(* IEC 61131-3 sources: STVM/tests/functional (part 2) *)

FUNCTION Scale_85 : REAL
VAR_INPUT
    raw : REAL;
END_VAR
    tmp_real := raw * 1.85;
    IF tmp_real > 10000.0 THEN
        tmp_real := 10000.0;
    END_IF;
    Scale_85 := tmp_real;
END_FUNCTION

FUNCTION LimitCheck_85 : BOOL
VAR_INPUT
    value : REAL;
    lo : REAL;
    hi : REAL;
END_VAR
    LimitCheck_85 := (value >= lo) AND (value <= hi);
END_FUNCTION

(* @LOOP_MAX(100) - 校验函数 86 *)
FUNCTION Verify_Channel_86 : INT
VAR_INPUT
    value : REAL;
    limit : REAL;
END_VAR
    tmp_bool := (value <= limit);
    IF tmp_bool THEN
        Verify_Channel_86 := 0;
    ELSE
        Verify_Channel_86 := -1;
    END_IF;
END_FUNCTION

FUNCTION Scale_86 : REAL
VAR_INPUT
    raw : REAL;
END_VAR
    tmp_real := raw * 1.86;
    IF tmp_real > 10000.0 THEN
        tmp_real := 10000.0;
    END_IF;
    Scale_86 := tmp_real;
END_FUNCTION

FUNCTION LimitCheck_86 : BOOL
VAR_INPUT
    value : REAL;
    lo : REAL;
    hi : REAL;
END_VAR
    LimitCheck_86 := (value >= lo) AND (value <= hi);
END_FUNCTION

(* @LOOP_MAX(100) - 校验函数 87 *)
FUNCTION Verify_Channel_87 : INT
VAR_INPUT
    value : REAL;
    limit : REAL;
END_VAR
    tmp_bool := (value <= limit);
    IF tmp_bool THEN
        Verify_Channel_87 := 0;
    ELSE
        Verify_Channel_87 := -1;
    END_IF;
END_FUNCTION

FUNCTION Scale_87 : REAL
VAR_INPUT
    raw : REAL;
END_VAR
    tmp_real := raw * 1.87;
    IF tmp_real > 10000.0 THEN
        tmp_real := 10000.0;
    END_IF;
    Scale_87 := tmp_real;
END_FUNCTION

FUNCTION LimitCheck_87 : BOOL
VAR_INPUT
    value : REAL;
    lo : REAL;
    hi : REAL;
END_VAR
    LimitCheck_87 := (value >= lo) AND (value <= hi);
END_FUNCTION

(* @LOOP_MAX(100) - 校验函数 88 *)
FUNCTION Verify_Channel_88 : INT
VAR_INPUT
    value : REAL;
    limit : REAL;
END_VAR
    tmp_bool := (value <= limit);
    IF tmp_bool THEN
        Verify_Channel_88 := 0;
    ELSE
        Verify_Channel_88 := -1;
    END_IF;
END_FUNCTION

FUNCTION Scale_88 : REAL
VAR_INPUT
    raw : REAL;
END_VAR
    tmp_real := raw * 1.88;
    IF tmp_real > 10000.0 THEN
        tmp_real := 10000.0;
    END_IF;
    Scale_88 := tmp_real;
END_FUNCTION

FUNCTION LimitCheck_88 : BOOL
VAR_INPUT
    value : REAL;
    lo : REAL;
    hi : REAL;
END_VAR
    LimitCheck_88 := (value >= lo) AND (value <= hi);
END_FUNCTION

(* @LOOP_MAX(100) - 校验函数 89 *)
FUNCTION Verify_Channel_89 : INT
VAR_INPUT
    value : REAL;
    limit : REAL;
END_VAR
    tmp_bool := (value <= limit);
    IF tmp_bool THEN
        Verify_Channel_89 := 0;
    ELSE
        Verify_Channel_89 := -1;
    END_IF;
END_FUNCTION

FUNCTION Scale_89 : REAL
VAR_INPUT
    raw : REAL;
END_VAR
    tmp_real := raw * 1.89;
    IF tmp_real > 10000.0 THEN
        tmp_real := 10000.0;
    END_IF;
    Scale_89 := tmp_real;
END_FUNCTION

FUNCTION LimitCheck_89 : BOOL
VAR_INPUT
    value : REAL;
    lo : REAL;
    hi : REAL;
END_VAR
    LimitCheck_89 := (value >= lo) AND (value <= hi);
END_FUNCTION

(* @LOOP_MAX(100) - 校验函数 90 *)
FUNCTION Verify_Channel_90 : INT
VAR_INPUT
    value : REAL;
    limit : REAL;
END_VAR
    tmp_bool := (value <= limit);
    IF tmp_bool THEN
        Verify_Channel_90 := 0;
    ELSE
        Verify_Channel_90 := -1;
    END_IF;
END_FUNCTION

FUNCTION Scale_90 : REAL
VAR_INPUT
    raw : REAL;
END_VAR
    tmp_real := raw * 1.90;
    IF tmp_real > 10000.0 THEN
        tmp_real := 10000.0;
    END_IF;
    Scale_90 := tmp_real;
END_FUNCTION

FUNCTION LimitCheck_90 : BOOL
VAR_INPUT
    value : REAL;
    lo : REAL;
    hi : REAL;
END_VAR
    LimitCheck_90 := (value >= lo) AND (value <= hi);
END_FUNCTION

(* @LOOP_MAX(100) - 校验函数 91 *)
FUNCTION Verify_Channel_91 : INT
VAR_INPUT
    value : REAL;
    limit : REAL;
END_VAR
    tmp_bool := (value <= limit);
    IF tmp_bool THEN
        Verify_Channel_91 := 0;
    ELSE
        Verify_Channel_91 := -1;
    END_IF;
END_FUNCTION

FUNCTION Scale_91 : REAL
VAR_INPUT
    raw : REAL;
END_VAR
    tmp_real := raw * 1.91;
    IF tmp_real > 10000.0 THEN
        tmp_real := 10000.0;
    END_IF;
    Scale_91 := tmp_real;
END_FUNCTION

FUNCTION LimitCheck_91 : BOOL
VAR_INPUT
    value : REAL;
    lo : REAL;
    hi : REAL;
END_VAR
    LimitCheck_91 := (value >= lo) AND (value <= hi);
END_FUNCTION

(* @LOOP_MAX(100) - 校验函数 92 *)
FUNCTION Verify_Channel_92 : INT
VAR_INPUT
    value : REAL;
    limit : REAL;
END_VAR
    tmp_bool := (value <= limit);
    IF tmp_bool THEN
        Verify_Channel_92 := 0;
    ELSE
        Verify_Channel_92 := -1;
    END_IF;
END_FUNCTION

FUNCTION Scale_92 : REAL
VAR_INPUT
    raw : REAL;
END_VAR
    tmp_real := raw * 1.92;
    IF tmp_real > 10000.0 THEN
        tmp_real := 10000.0;
    END_IF;
    Scale_92 := tmp_real;
END_FUNCTION

FUNCTION LimitCheck_92 : BOOL
VAR_INPUT
    value : REAL;
    lo : REAL;
    hi : REAL;
END_VAR
    LimitCheck_92 := (value >= lo) AND (value <= hi);
END_FUNCTION

(* @LOOP_MAX(100) - 校验函数 93 *)
FUNCTION Verify_Channel_93 : INT
VAR_INPUT
    value : REAL;
    limit : REAL;
END_VAR
    tmp_bool := (value <= limit);
    IF tmp_bool THEN
        Verify_Channel_93 := 0;
    ELSE
        Verify_Channel_93 := -1;
    END_IF;
END_FUNCTION

FUNCTION Scale_93 : REAL
VAR_INPUT
    raw : REAL;
END_VAR
    tmp_real := raw * 1.93;
    IF tmp_real > 10000.0 THEN
        tmp_real := 10000.0;
    END_IF;
    Scale_93 := tmp_real;
END_FUNCTION

FUNCTION LimitCheck_93 : BOOL
VAR_INPUT
    value : REAL;
    lo : REAL;
    hi : REAL;
END_VAR
    LimitCheck_93 := (value >= lo) AND (value <= hi);
END_FUNCTION

(* @LOOP_MAX(100) - 校验函数 94 *)
FUNCTION Verify_Channel_94 : INT
VAR_INPUT
    value : REAL;
    limit : REAL;
END_VAR
    tmp_bool := (value <= limit);
    IF tmp_bool THEN
        Verify_Channel_94 := 0;
    ELSE
        Verify_Channel_94 := -1;
    END_IF;
END_FUNCTION

FUNCTION Scale_94 : REAL
VAR_INPUT
    raw : REAL;
END_VAR
    tmp_real := raw * 1.94;
    IF tmp_real > 10000.0 THEN
        tmp_real := 10000.0;
    END_IF;
    Scale_94 := tmp_real;
END_FUNCTION

FUNCTION LimitCheck_94 : BOOL
VAR_INPUT
    value : REAL;
    lo : REAL;
    hi : REAL;
END_VAR
    LimitCheck_94 := (value >= lo) AND (value <= hi);
END_FUNCTION

(* @LOOP_MAX(100) - 校验函数 95 *)
FUNCTION Verify_Channel_95 : INT
VAR_INPUT
    value : REAL;
    limit : REAL;
END_VAR
    tmp_bool := (value <= limit);
    IF tmp_bool THEN
        Verify_Channel_95 := 0;
    ELSE
        Verify_Channel_95 := -1;
    END_IF;
END_FUNCTION

FUNCTION Scale_95 : REAL
VAR_INPUT
    raw : REAL;
END_VAR
    tmp_real := raw * 1.95;
    IF tmp_real > 10000.0 THEN
        tmp_real := 10000.0;
    END_IF;
    Scale_95 := tmp_real;
END_FUNCTION

FUNCTION LimitCheck_95 : BOOL
VAR_INPUT
    value : REAL;
    lo : REAL;
    hi : REAL;
END_VAR
    LimitCheck_95 := (value >= lo) AND (value <= hi);
END_FUNCTION

(* @LOOP_MAX(100) - 校验函数 96 *)
FUNCTION Verify_Channel_96 : INT
VAR_INPUT
    value : REAL;
    limit : REAL;
END_VAR
    tmp_bool := (value <= limit);
    IF tmp_bool THEN
        Verify_Channel_96 := 0;
    ELSE
        Verify_Channel_96 := -1;
    END_IF;
END_FUNCTION

FUNCTION Scale_96 : REAL
VAR_INPUT
    raw : REAL;
END_VAR
    tmp_real := raw * 1.96;
    IF tmp_real > 10000.0 THEN
        tmp_real := 10000.0;
    END_IF;
    Scale_96 := tmp_real;
END_FUNCTION

FUNCTION LimitCheck_96 : BOOL
VAR_INPUT
    value : REAL;
    lo : REAL;
    hi : REAL;
END_VAR
    LimitCheck_96 := (value >= lo) AND (value <= hi);
END_FUNCTION

(* @LOOP_MAX(100) - 校验函数 97 *)
FUNCTION Verify_Channel_97 : INT
VAR_INPUT
    value : REAL;
    limit : REAL;
END_VAR
    tmp_bool := (value <= limit);
    IF tmp_bool THEN
        Verify_Channel_97 := 0;
    ELSE
        Verify_Channel_97 := -1;
    END_IF;
END_FUNCTION

FUNCTION Scale_97 : REAL
VAR_INPUT
    raw : REAL;
END_VAR
    tmp_real := raw * 1.97;
    IF tmp_real > 10000.0 THEN
        tmp_real := 10000.0;
    END_IF;
    Scale_97 := tmp_real;
END_FUNCTION

FUNCTION LimitCheck_97 : BOOL
VAR_INPUT
    value : REAL;
    lo : REAL;
    hi : REAL;
END_VAR
    LimitCheck_97 := (value >= lo) AND (value <= hi);
END_FUNCTION

(* @LOOP_MAX(100) - 校验函数 98 *)
FUNCTION Verify_Channel_98 : INT
VAR_INPUT
    value : REAL;
    limit : REAL;
END_VAR
    tmp_bool := (value <= limit);
    IF tmp_bool THEN
        Verify_Channel_98 := 0;
    ELSE
        Verify_Channel_98 := -1;
    END_IF;
END_FUNCTION

FUNCTION Scale_98 : REAL
VAR_INPUT
    raw : REAL;
END_VAR
    tmp_real := raw * 1.98;
    IF tmp_real > 10000.0 THEN
        tmp_real := 10000.0;
    END_IF;
    Scale_98 := tmp_real;
END_FUNCTION

FUNCTION LimitCheck_98 : BOOL
VAR_INPUT
    value : REAL;
    lo : REAL;
    hi : REAL;
END_VAR
    LimitCheck_98 := (value >= lo) AND (value <= hi);
END_FUNCTION

(* @LOOP_MAX(100) - 校验函数 99 *)
FUNCTION Verify_Channel_99 : INT
VAR_INPUT
    value : REAL;
    limit : REAL;
END_VAR
    tmp_bool := (value <= limit);
    IF tmp_bool THEN
        Verify_Channel_99 := 0;
    ELSE
        Verify_Channel_99 := -1;
    END_IF;
END_FUNCTION

FUNCTION Scale_99 : REAL
VAR_INPUT
    raw : REAL;
END_VAR
    tmp_real := raw * 1.99;
    IF tmp_real > 10000.0 THEN
        tmp_real := 10000.0;
    END_IF;
    Scale_99 := tmp_real;
END_FUNCTION

FUNCTION LimitCheck_99 : BOOL
VAR_INPUT
    value : REAL;
    lo : REAL;
    hi : REAL;
END_VAR
    LimitCheck_99 := (value >= lo) AND (value <= hi);
END_FUNCTION

(* @LOOP_MAX(100) - 校验函数 100 *)
FUNCTION Verify_Channel_100 : INT
VAR_INPUT
    value : REAL;
    limit : REAL;
END_VAR
    tmp_bool := (value <= limit);
    IF tmp_bool THEN
        Verify_Channel_100 := 0;
    ELSE
        Verify_Channel_100 := -1;
    END_IF;
END_FUNCTION

FUNCTION Scale_100 : REAL
VAR_INPUT
    raw : REAL;
END_VAR
    tmp_real := raw * 1.100;
    IF tmp_real > 10000.0 THEN
        tmp_real := 10000.0;
    END_IF;
    Scale_100 := tmp_real;
END_FUNCTION

FUNCTION LimitCheck_100 : BOOL
VAR_INPUT
    value : REAL;
    lo : REAL;
    hi : REAL;
END_VAR
    LimitCheck_100 := (value >= lo) AND (value <= hi);
END_FUNCTION

(* @LOOP_MAX(100) - 校验函数 101 *)
FUNCTION Verify_Channel_101 : INT
VAR_INPUT
    value : REAL;
    limit : REAL;
END_VAR
    tmp_bool := (value <= limit);
    IF tmp_bool THEN
        Verify_Channel_101 := 0;
    ELSE
        Verify_Channel_101 := -1;
    END_IF;
END_FUNCTION

FUNCTION Scale_101 : REAL
VAR_INPUT
    raw : REAL;
END_VAR
    tmp_real := raw * 1.101;
    IF tmp_real > 10000.0 THEN
        tmp_real := 10000.0;
    END_IF;
    Scale_101 := tmp_real;
END_FUNCTION

FUNCTION LimitCheck_101 : BOOL
VAR_INPUT
    value : REAL;
    lo : REAL;
    hi : REAL;
END_VAR
    LimitCheck_101 := (value >= lo) AND (value <= hi);
END_FUNCTION

(* @LOOP_MAX(100) - 校验函数 102 *)
FUNCTION Verify_Channel_102 : INT
VAR_INPUT
    value : REAL;
    limit : REAL;
END_VAR
    tmp_bool := (value <= limit);
    IF tmp_bool THEN
        Verify_Channel_102 := 0;
    ELSE
        Verify_Channel_102 := -1;
    END_IF;
END_FUNCTION

FUNCTION Scale_102 : REAL
VAR_INPUT
    raw : REAL;
END_VAR
    tmp_real := raw * 1.102;
    IF tmp_real > 10000.0 THEN
        tmp_real := 10000.0;
    END_IF;
    Scale_102 := tmp_real;
END_FUNCTION

FUNCTION LimitCheck_102 : BOOL
VAR_INPUT
    value : REAL;
    lo : REAL;
    hi : REAL;
END_VAR
    LimitCheck_102 := (value >= lo) AND (value <= hi);
END_FUNCTION

(* @LOOP_MAX(100) - 校验函数 103 *)
FUNCTION Verify_Channel_103 : INT
VAR_INPUT
    value : REAL;
    limit : REAL;
END_VAR
    tmp_bool := (value <= limit);
    IF tmp_bool THEN
        Verify_Channel_103 := 0;
    ELSE
        Verify_Channel_103 := -1;
    END_IF;
END_FUNCTION

FUNCTION Scale_103 : REAL
VAR_INPUT
    raw : REAL;
END_VAR
    tmp_real := raw * 1.103;
    IF tmp_real > 10000.0 THEN
        tmp_real := 10000.0;
    END_IF;
    Scale_103 := tmp_real;
END_FUNCTION

FUNCTION LimitCheck_103 : BOOL
VAR_INPUT
    value : REAL;
    lo : REAL;
    hi : REAL;
END_VAR
    LimitCheck_103 := (value >= lo) AND (value <= hi);
END_FUNCTION

(* @LOOP_MAX(100) - 校验函数 104 *)
FUNCTION Verify_Channel_104 : INT
VAR_INPUT
    value : REAL;
    limit : REAL;
END_VAR
    tmp_bool := (value <= limit);
    IF tmp_bool THEN
        Verify_Channel_104 := 0;
    ELSE
        Verify_Channel_104 := -1;
    END_IF;
END_FUNCTION

FUNCTION Scale_104 : REAL
VAR_INPUT
    raw : REAL;
END_VAR
    tmp_real := raw * 1.104;
    IF tmp_real > 10000.0 THEN
        tmp_real := 10000.0;
    END_IF;
    Scale_104 := tmp_real;
END_FUNCTION

FUNCTION LimitCheck_104 : BOOL
VAR_INPUT
    value : REAL;
    lo : REAL;
    hi : REAL;
END_VAR
    LimitCheck_104 := (value >= lo) AND (value <= hi);
END_FUNCTION

(* @LOOP_MAX(100) - 校验函数 105 *)
FUNCTION Verify_Channel_105 : INT
VAR_INPUT
    value : REAL;
    limit : REAL;
END_VAR
    tmp_bool := (value <= limit);
    IF tmp_bool THEN
        Verify_Channel_105 := 0;
    ELSE
        Verify_Channel_105 := -1;
    END_IF;
END_FUNCTION

FUNCTION Scale_105 : REAL
VAR_INPUT
    raw : REAL;
END_VAR
    tmp_real := raw * 1.105;
    IF tmp_real > 10000.0 THEN
        tmp_real := 10000.0;
    END_IF;
    Scale_105 := tmp_real;
END_FUNCTION

FUNCTION LimitCheck_105 : BOOL
VAR_INPUT
    value : REAL;
    lo : REAL;
    hi : REAL;
END_VAR
    LimitCheck_105 := (value >= lo) AND (value <= hi);
END_FUNCTION

(* @LOOP_MAX(100) - 校验函数 106 *)
FUNCTION Verify_Channel_106 : INT
VAR_INPUT
    value : REAL;
    limit : REAL;
END_VAR
    tmp_bool := (value <= limit);
    IF tmp_bool THEN
        Verify_Channel_106 := 0;
    ELSE
        Verify_Channel_106 := -1;
    END_IF;
END_FUNCTION

FUNCTION Scale_106 : REAL
VAR_INPUT
    raw : REAL;
END_VAR
    tmp_real := raw * 1.106;
    IF tmp_real > 10000.0 THEN
        tmp_real := 10000.0;
    END_IF;
    Scale_106 := tmp_real;
END_FUNCTION

FUNCTION LimitCheck_106 : BOOL
VAR_INPUT
    value : REAL;
    lo : REAL;
    hi : REAL;
END_VAR
    LimitCheck_106 := (value >= lo) AND (value <= hi);
END_FUNCTION

(* @LOOP_MAX(100) - 校验函数 107 *)
FUNCTION Verify_Channel_107 : INT
VAR_INPUT
    value : REAL;
    limit : REAL;
END_VAR
    tmp_bool := (value <= limit);
    IF tmp_bool THEN
        Verify_Channel_107 := 0;
    ELSE
        Verify_Channel_107 := -1;
    END_IF;
END_FUNCTION

FUNCTION Scale_107 : REAL
VAR_INPUT
    raw : REAL;
END_VAR
    tmp_real := raw * 1.107;
    IF tmp_real > 10000.0 THEN
        tmp_real := 10000.0;
    END_IF;
    Scale_107 := tmp_real;
END_FUNCTION

FUNCTION LimitCheck_107 : BOOL
VAR_INPUT
    value : REAL;
    lo : REAL;
    hi : REAL;
END_VAR
    LimitCheck_107 := (value >= lo) AND (value <= hi);
END_FUNCTION

(* @LOOP_MAX(100) - 校验函数 108 *)
FUNCTION Verify_Channel_108 : INT
VAR_INPUT
    value : REAL;
    limit : REAL;
END_VAR
    tmp_bool := (value <= limit);
    IF tmp_bool THEN
        Verify_Channel_108 := 0;
    ELSE
        Verify_Channel_108 := -1;
    END_IF;
END_FUNCTION

FUNCTION Scale_108 : REAL
VAR_INPUT
    raw : REAL;
END_VAR
    tmp_real := raw * 1.108;
    IF tmp_real > 10000.0 THEN
        tmp_real := 10000.0;
    END_IF;
    Scale_108 := tmp_real;
END_FUNCTION

FUNCTION LimitCheck_108 : BOOL
VAR_INPUT
    value : REAL;
    lo : REAL;
    hi : REAL;
END_VAR
    LimitCheck_108 := (value >= lo) AND (value <= hi);
END_FUNCTION

(* @LOOP_MAX(100) - 校验函数 109 *)
FUNCTION Verify_Channel_109 : INT
VAR_INPUT
    value : REAL;
    limit : REAL;
END_VAR
    tmp_bool := (value <= limit);
    IF tmp_bool THEN
        Verify_Channel_109 := 0;
    ELSE
        Verify_Channel_109 := -1;
    END_IF;
END_FUNCTION

FUNCTION Scale_109 : REAL
VAR_INPUT
    raw : REAL;
END_VAR
    tmp_real := raw * 1.109;
    IF tmp_real > 10000.0 THEN
        tmp_real := 10000.0;
    END_IF;
    Scale_109 := tmp_real;
END_FUNCTION

FUNCTION LimitCheck_109 : BOOL
VAR_INPUT
    value : REAL;
    lo : REAL;
    hi : REAL;
END_VAR
    LimitCheck_109 := (value >= lo) AND (value <= hi);
END_FUNCTION

(* @LOOP_MAX(100) - 校验函数 110 *)
FUNCTION Verify_Channel_110 : INT
VAR_INPUT
    value : REAL;
    limit : REAL;
END_VAR
    tmp_bool := (value <= limit);
    IF tmp_bool THEN
        Verify_Channel_110 := 0;
    ELSE
        Verify_Channel_110 := -1;
    END_IF;
END_FUNCTION

FUNCTION Scale_110 : REAL
VAR_INPUT
    raw : REAL;
END_VAR
    tmp_real := raw * 1.110;
    IF tmp_real > 10000.0 THEN
        tmp_real := 10000.0;
    END_IF;
    Scale_110 := tmp_real;
END_FUNCTION

FUNCTION LimitCheck_110 : BOOL
VAR_INPUT
    value : REAL;
    lo : REAL;
    hi : REAL;
END_VAR
    LimitCheck_110 := (value >= lo) AND (value <= hi);
END_FUNCTION

(* @LOOP_MAX(100) - 校验函数 111 *)
FUNCTION Verify_Channel_111 : INT
VAR_INPUT
    value : REAL;
    limit : REAL;
END_VAR
    tmp_bool := (value <= limit);
    IF tmp_bool THEN
        Verify_Channel_111 := 0;
    ELSE
        Verify_Channel_111 := -1;
    END_IF;
END_FUNCTION

FUNCTION Scale_111 : REAL
VAR_INPUT
    raw : REAL;
END_VAR
    tmp_real := raw * 1.111;
    IF tmp_real > 10000.0 THEN
        tmp_real := 10000.0;
    END_IF;
    Scale_111 := tmp_real;
END_FUNCTION

FUNCTION LimitCheck_111 : BOOL
VAR_INPUT
    value : REAL;
    lo : REAL;
    hi : REAL;
END_VAR
    LimitCheck_111 := (value >= lo) AND (value <= hi);
END_FUNCTION

(* @LOOP_MAX(100) - 校验函数 112 *)
FUNCTION Verify_Channel_112 : INT
VAR_INPUT
    value : REAL;
    limit : REAL;
END_VAR
    tmp_bool := (value <= limit);
    IF tmp_bool THEN
        Verify_Channel_112 := 0;
    ELSE
        Verify_Channel_112 := -1;
    END_IF;
END_FUNCTION

FUNCTION Scale_112 : REAL
VAR_INPUT
    raw : REAL;
END_VAR
    tmp_real := raw * 1.112;
    IF tmp_real > 10000.0 THEN
        tmp_real := 10000.0;
    END_IF;
    Scale_112 := tmp_real;
END_FUNCTION

FUNCTION LimitCheck_112 : BOOL
VAR_INPUT
    value : REAL;
    lo : REAL;
    hi : REAL;
END_VAR
    LimitCheck_112 := (value >= lo) AND (value <= hi);
END_FUNCTION

(* @LOOP_MAX(100) - 校验函数 113 *)
FUNCTION Verify_Channel_113 : INT
VAR_INPUT
    value : REAL;
    limit : REAL;
END_VAR
    tmp_bool := (value <= limit);
    IF tmp_bool THEN
        Verify_Channel_113 := 0;
    ELSE
        Verify_Channel_113 := -1;
    END_IF;
END_FUNCTION

FUNCTION Scale_113 : REAL
VAR_INPUT
    raw : REAL;
END_VAR
    tmp_real := raw * 1.113;
    IF tmp_real > 10000.0 THEN
        tmp_real := 10000.0;
    END_IF;
    Scale_113 := tmp_real;
END_FUNCTION

FUNCTION LimitCheck_113 : BOOL
VAR_INPUT
    value : REAL;
    lo : REAL;
    hi : REAL;
END_VAR
    LimitCheck_113 := (value >= lo) AND (value <= hi);
END_FUNCTION

(* @LOOP_MAX(100) - 校验函数 114 *)
FUNCTION Verify_Channel_114 : INT
VAR_INPUT
    value : REAL;
    limit : REAL;
END_VAR
    tmp_bool := (value <= limit);
    IF tmp_bool THEN
        Verify_Channel_114 := 0;
    ELSE
        Verify_Channel_114 := -1;
    END_IF;
END_FUNCTION

FUNCTION Scale_114 : REAL
VAR_INPUT
    raw : REAL;
END_VAR
    tmp_real := raw * 1.114;
    IF tmp_real > 10000.0 THEN
        tmp_real := 10000.0;
    END_IF;
    Scale_114 := tmp_real;
END_FUNCTION

FUNCTION LimitCheck_114 : BOOL
VAR_INPUT
    value : REAL;
    lo : REAL;
    hi : REAL;
END_VAR
    LimitCheck_114 := (value >= lo) AND (value <= hi);
END_FUNCTION

(* @LOOP_MAX(100) - 校验函数 115 *)
FUNCTION Verify_Channel_115 : INT
VAR_INPUT
    value : REAL;
    limit : REAL;
END_VAR
    tmp_bool := (value <= limit);
    IF tmp_bool THEN
        Verify_Channel_115 := 0;
    ELSE
        Verify_Channel_115 := -1;
    END_IF;
END_FUNCTION

FUNCTION Scale_115 : REAL
VAR_INPUT
    raw : REAL;
END_VAR
    tmp_real := raw * 1.115;
    IF tmp_real > 10000.0 THEN
        tmp_real := 10000.0;
    END_IF;
    Scale_115 := tmp_real;
END_FUNCTION

FUNCTION LimitCheck_115 : BOOL
VAR_INPUT
    value : REAL;
    lo : REAL;
    hi : REAL;
END_VAR
    LimitCheck_115 := (value >= lo) AND (value <= hi);
END_FUNCTION

(* @LOOP_MAX(100) - 校验函数 116 *)
FUNCTION Verify_Channel_116 : INT
VAR_INPUT
    value : REAL;
    limit : REAL;
END_VAR
    tmp_bool := (value <= limit);
    IF tmp_bool THEN
        Verify_Channel_116 := 0;
    ELSE
        Verify_Channel_116 := -1;
    END_IF;
END_FUNCTION

FUNCTION Scale_116 : REAL
VAR_INPUT
    raw : REAL;
END_VAR
    tmp_real := raw * 1.116;
    IF tmp_real > 10000.0 THEN
        tmp_real := 10000.0;
    END_IF;
    Scale_116 := tmp_real;
END_FUNCTION

FUNCTION LimitCheck_116 : BOOL
VAR_INPUT
    value : REAL;
    lo : REAL;
    hi : REAL;
END_VAR
    LimitCheck_116 := (value >= lo) AND (value <= hi);
END_FUNCTION

(* @LOOP_MAX(100) - 校验函数 117 *)
FUNCTION Verify_Channel_117 : INT
VAR_INPUT
    value : REAL;
    limit : REAL;
END_VAR
    tmp_bool := (value <= limit);
    IF tmp_bool THEN
        Verify_Channel_117 := 0;
    ELSE
        Verify_Channel_117 := -1;
    END_IF;
END_FUNCTION

FUNCTION Scale_117 : REAL
VAR_INPUT
    raw : REAL;
END_VAR
    tmp_real := raw * 1.117;
    IF tmp_real > 10000.0 THEN
        tmp_real := 10000.0;
    END_IF;
    Scale_117 := tmp_real;
END_FUNCTION

FUNCTION LimitCheck_117 : BOOL
VAR_INPUT
    value : REAL;
    lo : REAL;
    hi : REAL;
END_VAR
    LimitCheck_117 := (value >= lo) AND (value <= hi);
END_FUNCTION

(* @LOOP_MAX(100) - 校验函数 118 *)
FUNCTION Verify_Channel_118 : INT
VAR_INPUT
    value : REAL;
    limit : REAL;
END_VAR
    tmp_bool := (value <= limit);
    IF tmp_bool THEN
        Verify_Channel_118 := 0;
    ELSE
        Verify_Channel_118 := -1;
    END_IF;
END_FUNCTION

FUNCTION Scale_118 : REAL
VAR_INPUT
    raw : REAL;
END_VAR
    tmp_real := raw * 1.118;
    IF tmp_real > 10000.0 THEN
        tmp_real := 10000.0;
    END_IF;
    Scale_118 := tmp_real;
END_FUNCTION

FUNCTION LimitCheck_118 : BOOL
VAR_INPUT
    value : REAL;
    lo : REAL;
    hi : REAL;
END_VAR
    LimitCheck_118 := (value >= lo) AND (value <= hi);
END_FUNCTION

(* @LOOP_MAX(100) - 校验函数 119 *)
FUNCTION Verify_Channel_119 : INT
VAR_INPUT
    value : REAL;
    limit : REAL;
END_VAR
    tmp_bool := (value <= limit);
    IF tmp_bool THEN
        Verify_Channel_119 := 0;
    ELSE
        Verify_Channel_119 := -1;
    END_IF;
END_FUNCTION

FUNCTION Scale_119 : REAL
VAR_INPUT
    raw : REAL;
END_VAR
    tmp_real := raw * 1.119;
    IF tmp_real > 10000.0 THEN
        tmp_real := 10000.0;
    END_IF;
    Scale_119 := tmp_real;
END_FUNCTION

FUNCTION LimitCheck_119 : BOOL
VAR_INPUT
    value : REAL;
    lo : REAL;
    hi : REAL;
END_VAR
    LimitCheck_119 := (value >= lo) AND (value <= hi);
END_FUNCTION

(* @LOOP_MAX(100) - 校验函数 120 *)
FUNCTION Verify_Channel_120 : INT
VAR_INPUT
    value : REAL;
    limit : REAL;
END_VAR
    tmp_bool := (value <= limit);
    IF tmp_bool THEN
        Verify_Channel_120 := 0;
    ELSE
        Verify_Channel_120 := -1;
    END_IF;
END_FUNCTION

FUNCTION Scale_120 : REAL
VAR_INPUT
    raw : REAL;
END_VAR
    tmp_real := raw * 1.120;
    IF tmp_real > 10000.0 THEN
        tmp_real := 10000.0;
    END_IF;
    Scale_120 := tmp_real;
END_FUNCTION

FUNCTION LimitCheck_120 : BOOL
VAR_INPUT
    value : REAL;
    lo : REAL;
    hi : REAL;
END_VAR
    LimitCheck_120 := (value >= lo) AND (value <= hi);
END_FUNCTION

(* @LOOP_MAX(100) - 校验函数 121 *)
FUNCTION Verify_Channel_121 : INT
VAR_INPUT
    value : REAL;
    limit : REAL;
END_VAR
    tmp_bool := (value <= limit);
    IF tmp_bool THEN
        Verify_Channel_121 := 0;
    ELSE
        Verify_Channel_121 := -1;
    END_IF;
END_FUNCTION

FUNCTION Scale_121 : REAL
VAR_INPUT
    raw : REAL;
END_VAR
    tmp_real := raw * 1.121;
    IF tmp_real > 10000.0 THEN
        tmp_real := 10000.0;
    END_IF;
    Scale_121 := tmp_real;
END_FUNCTION

FUNCTION LimitCheck_121 : BOOL
VAR_INPUT
    value : REAL;
    lo : REAL;
    hi : REAL;
END_VAR
    LimitCheck_121 := (value >= lo) AND (value <= hi);
END_FUNCTION

(* @LOOP_MAX(100) - 校验函数 122 *)
FUNCTION Verify_Channel_122 : INT
VAR_INPUT
    value : REAL;
    limit : REAL;
END_VAR
    tmp_bool := (value <= limit);
    IF tmp_bool THEN
        Verify_Channel_122 := 0;
    ELSE
        Verify_Channel_122 := -1;
    END_IF;
END_FUNCTION

FUNCTION Scale_122 : REAL
VAR_INPUT
    raw : REAL;
END_VAR
    tmp_real := raw * 1.122;
    IF tmp_real > 10000.0 THEN
        tmp_real := 10000.0;
    END_IF;
    Scale_122 := tmp_real;
END_FUNCTION

FUNCTION LimitCheck_122 : BOOL
VAR_INPUT
    value : REAL;
    lo : REAL;
    hi : REAL;
END_VAR
    LimitCheck_122 := (value >= lo) AND (value <= hi);
END_FUNCTION

(* @LOOP_MAX(100) - 校验函数 123 *)
FUNCTION Verify_Channel_123 : INT
VAR_INPUT
    value : REAL;
    limit : REAL;
END_VAR
    tmp_bool := (value <= limit);
    IF tmp_bool THEN
        Verify_Channel_123 := 0;
    ELSE
        Verify_Channel_123 := -1;
    END_IF;
END_FUNCTION

FUNCTION Scale_123 : REAL
VAR_INPUT
    raw : REAL;
END_VAR
    tmp_real := raw * 1.123;
    IF tmp_real > 10000.0 THEN
        tmp_real := 10000.0;
    END_IF;
    Scale_123 := tmp_real;
END_FUNCTION

FUNCTION LimitCheck_123 : BOOL
VAR_INPUT
    value : REAL;
    lo : REAL;
    hi : REAL;
END_VAR
    LimitCheck_123 := (value >= lo) AND (value <= hi);
END_FUNCTION

(* @LOOP_MAX(100) - 校验函数 124 *)
FUNCTION Verify_Channel_124 : INT
VAR_INPUT
    value : REAL;
    limit : REAL;
END_VAR
    tmp_bool := (value <= limit);
    IF tmp_bool THEN
        Verify_Channel_124 := 0;
    ELSE
        Verify_Channel_124 := -1;
    END_IF;
END_FUNCTION

FUNCTION Scale_124 : REAL
VAR_INPUT
    raw : REAL;
END_VAR
    tmp_real := raw * 1.124;
    IF tmp_real > 10000.0 THEN
        tmp_real := 10000.0;
    END_IF;
    Scale_124 := tmp_real;
END_FUNCTION

FUNCTION LimitCheck_124 : BOOL
VAR_INPUT
    value : REAL;
    lo : REAL;
    hi : REAL;
END_VAR
    LimitCheck_124 := (value >= lo) AND (value <= hi);
END_FUNCTION

(* @LOOP_MAX(100) - 校验函数 125 *)
FUNCTION Verify_Channel_125 : INT
VAR_INPUT
    value : REAL;
    limit : REAL;
END_VAR
    tmp_bool := (value <= limit);
    IF tmp_bool THEN
        Verify_Channel_125 := 0;
    ELSE
        Verify_Channel_125 := -1;
    END_IF;
END_FUNCTION

FUNCTION Scale_125 : REAL
VAR_INPUT
    raw : REAL;
END_VAR
    tmp_real := raw * 1.125;
    IF tmp_real > 10000.0 THEN
        tmp_real := 10000.0;
    END_IF;
    Scale_125 := tmp_real;
END_FUNCTION

FUNCTION LimitCheck_125 : BOOL
VAR_INPUT
    value : REAL;
    lo : REAL;
    hi : REAL;
END_VAR
    LimitCheck_125 := (value >= lo) AND (value <= hi);
END_FUNCTION

(* @LOOP_MAX(100) - 校验函数 126 *)
FUNCTION Verify_Channel_126 : INT
VAR_INPUT
    value : REAL;
    limit : REAL;
END_VAR
    tmp_bool := (value <= limit);
    IF tmp_bool THEN
        Verify_Channel_126 := 0;
    ELSE
        Verify_Channel_126 := -1;
    END_IF;
END_FUNCTION

FUNCTION Scale_126 : REAL
VAR_INPUT
    raw : REAL;
END_VAR
    tmp_real := raw * 1.126;
    IF tmp_real > 10000.0 THEN
        tmp_real := 10000.0;
    END_IF;
    Scale_126 := tmp_real;
END_FUNCTION

FUNCTION LimitCheck_126 : BOOL
VAR_INPUT
    value : REAL;
    lo : REAL;
    hi : REAL;
END_VAR
    LimitCheck_126 := (value >= lo) AND (value <= hi);
END_FUNCTION

(* @LOOP_MAX(100) - 校验函数 127 *)
FUNCTION Verify_Channel_127 : INT
VAR_INPUT
    value : REAL;
    limit : REAL;
END_VAR
    tmp_bool := (value <= limit);
    IF tmp_bool THEN
        Verify_Channel_127 := 0;
    ELSE
        Verify_Channel_127 := -1;
    END_IF;
END_FUNCTION

FUNCTION Scale_127 : REAL
VAR_INPUT
    raw : REAL;
END_VAR
    tmp_real := raw * 1.127;
    IF tmp_real > 10000.0 THEN
        tmp_real := 10000.0;
    END_IF;
    Scale_127 := tmp_real;
END_FUNCTION

FUNCTION LimitCheck_127 : BOOL
VAR_INPUT
    value : REAL;
    lo : REAL;
    hi : REAL;
END_VAR
    LimitCheck_127 := (value >= lo) AND (value <= hi);
END_FUNCTION

(* @LOOP_MAX(100) - 校验函数 128 *)
FUNCTION Verify_Channel_128 : INT
VAR_INPUT
    value : REAL;
    limit : REAL;
END_VAR
    tmp_bool := (value <= limit);
    IF tmp_bool THEN
        Verify_Channel_128 := 0;
    ELSE
        Verify_Channel_128 := -1;
    END_IF;
END_FUNCTION

FUNCTION Scale_128 : REAL
VAR_INPUT
    raw : REAL;
END_VAR
    tmp_real := raw * 1.128;
    IF tmp_real > 10000.0 THEN
        tmp_real := 10000.0;
    END_IF;
    Scale_128 := tmp_real;
END_FUNCTION

FUNCTION LimitCheck_128 : BOOL
VAR_INPUT
    value : REAL;
    lo : REAL;
    hi : REAL;
END_VAR
    LimitCheck_128 := (value >= lo) AND (value <= hi);
END_FUNCTION

(* @LOOP_MAX(100) - 校验函数 129 *)
FUNCTION Verify_Channel_129 : INT
VAR_INPUT
    value : REAL;
    limit : REAL;
END_VAR
    tmp_bool := (value <= limit);
    IF tmp_bool THEN
        Verify_Channel_129 := 0;
    ELSE
        Verify_Channel_129 := -1;
    END_IF;
END_FUNCTION

FUNCTION Scale_129 : REAL
VAR_INPUT
    raw : REAL;
END_VAR
    tmp_real := raw * 1.129;
    IF tmp_real > 10000.0 THEN
        tmp_real := 10000.0;
    END_IF;
    Scale_129 := tmp_real;
END_FUNCTION

FUNCTION LimitCheck_129 : BOOL
VAR_INPUT
    value : REAL;
    lo : REAL;
    hi : REAL;
END_VAR
    LimitCheck_129 := (value >= lo) AND (value <= hi);
END_FUNCTION

(* @LOOP_MAX(100) - 校验函数 130 *)
FUNCTION Verify_Channel_130 : INT
VAR_INPUT
    value : REAL;
    limit : REAL;
END_VAR
    tmp_bool := (value <= limit);
    IF tmp_bool THEN
        Verify_Channel_130 := 0;
    ELSE
        Verify_Channel_130 := -1;
    END_IF;
END_FUNCTION

FUNCTION Scale_130 : REAL
VAR_INPUT
    raw : REAL;
END_VAR
    tmp_real := raw * 1.130;
    IF tmp_real > 10000.0 THEN
        tmp_real := 10000.0;
    END_IF;
    Scale_130 := tmp_real;
END_FUNCTION

FUNCTION LimitCheck_130 : BOOL
VAR_INPUT
    value : REAL;
    lo : REAL;
    hi : REAL;
END_VAR
    LimitCheck_130 := (value >= lo) AND (value <= hi);
END_FUNCTION

(* @LOOP_MAX(100) - 校验函数 131 *)
FUNCTION Verify_Channel_131 : INT
VAR_INPUT
    value : REAL;
    limit : REAL;
END_VAR
    tmp_bool := (value <= limit);
    IF tmp_bool THEN
        Verify_Channel_131 := 0;
    ELSE
        Verify_Channel_131 := -1;
    END_IF;
END_FUNCTION

FUNCTION Scale_131 : REAL
VAR_INPUT
    raw : REAL;
END_VAR
    tmp_real := raw * 1.131;
    IF tmp_real > 10000.0 THEN
        tmp_real := 10000.0;
    END_IF;
    Scale_131 := tmp_real;
END_FUNCTION

FUNCTION LimitCheck_131 : BOOL
VAR_INPUT
    value : REAL;
    lo : REAL;
    hi : REAL;
END_VAR
    LimitCheck_131 := (value >= lo) AND (value <= hi);
END_FUNCTION

(* @LOOP_MAX(100) - 校验函数 132 *)
FUNCTION Verify_Channel_132 : INT
VAR_INPUT
    value : REAL;
    limit : REAL;
END_VAR
    tmp_bool := (value <= limit);
    IF tmp_bool THEN
        Verify_Channel_132 := 0;
    ELSE
        Verify_Channel_132 := -1;
    END_IF;
END_FUNCTION

FUNCTION Scale_132 : REAL
VAR_INPUT
    raw : REAL;
END_VAR
    tmp_real := raw * 1.132;
    IF tmp_real > 10000.0 THEN
        tmp_real := 10000.0;
    END_IF;
    Scale_132 := tmp_real;
END_FUNCTION

FUNCTION LimitCheck_132 : BOOL
VAR_INPUT
    value : REAL;
    lo : REAL;
    hi : REAL;
END_VAR
    LimitCheck_132 := (value >= lo) AND (value <= hi);
END_FUNCTION

(* @LOOP_MAX(100) - 校验函数 133 *)
FUNCTION Verify_Channel_133 : INT
VAR_INPUT
    value : REAL;
    limit : REAL;
END_VAR
    tmp_bool := (value <= limit);
    IF tmp_bool THEN
        Verify_Channel_133 := 0;
    ELSE
        Verify_Channel_133 := -1;
    END_IF;
END_FUNCTION

FUNCTION Scale_133 : REAL
VAR_INPUT
    raw : REAL;
END_VAR
    tmp_real := raw * 1.133;
    IF tmp_real > 10000.0 THEN
        tmp_real := 10000.0;
    END_IF;
    Scale_133 := tmp_real;
END_FUNCTION

FUNCTION LimitCheck_133 : BOOL
VAR_INPUT
    value : REAL;
    lo : REAL;
    hi : REAL;
END_VAR
    LimitCheck_133 := (value >= lo) AND (value <= hi);
END_FUNCTION

(* @LOOP_MAX(100) - 校验函数 134 *)
FUNCTION Verify_Channel_134 : INT
VAR_INPUT
    value : REAL;
    limit : REAL;
END_VAR
    tmp_bool := (value <= limit);
    IF tmp_bool THEN
        Verify_Channel_134 := 0;
    ELSE
        Verify_Channel_134 := -1;
    END_IF;
END_FUNCTION

FUNCTION Scale_134 : REAL
VAR_INPUT
    raw : REAL;
END_VAR
    tmp_real := raw * 1.134;
    IF tmp_real > 10000.0 THEN
        tmp_real := 10000.0;
    END_IF;
    Scale_134 := tmp_real;
END_FUNCTION

FUNCTION LimitCheck_134 : BOOL
VAR_INPUT
    value : REAL;
    lo : REAL;
    hi : REAL;
END_VAR
    LimitCheck_134 := (value >= lo) AND (value <= hi);
END_FUNCTION

(* @LOOP_MAX(100) - 校验函数 135 *)
FUNCTION Verify_Channel_135 : INT
VAR_INPUT
    value : REAL;
    limit : REAL;
END_VAR
    tmp_bool := (value <= limit);
    IF tmp_bool THEN
        Verify_Channel_135 := 0;
    ELSE
        Verify_Channel_135 := -1;
    END_IF;
END_FUNCTION

FUNCTION Scale_135 : REAL
VAR_INPUT
    raw : REAL;
END_VAR
    tmp_real := raw * 1.135;
    IF tmp_real > 10000.0 THEN
        tmp_real := 10000.0;
    END_IF;
    Scale_135 := tmp_real;
END_FUNCTION

FUNCTION LimitCheck_135 : BOOL
VAR_INPUT
    value : REAL;
    lo : REAL;
    hi : REAL;
END_VAR
    LimitCheck_135 := (value >= lo) AND (value <= hi);
END_FUNCTION

(* @LOOP_MAX(100) - 校验函数 136 *)
FUNCTION Verify_Channel_136 : INT
VAR_INPUT
    value : REAL;
    limit : REAL;
END_VAR
    tmp_bool := (value <= limit);
    IF tmp_bool THEN
        Verify_Channel_136 := 0;
    ELSE
        Verify_Channel_136 := -1;
    END_IF;
END_FUNCTION

FUNCTION Scale_136 : REAL
VAR_INPUT
    raw : REAL;
END_VAR
    tmp_real := raw * 1.136;
    IF tmp_real > 10000.0 THEN
        tmp_real := 10000.0;
    END_IF;
    Scale_136 := tmp_real;
END_FUNCTION

FUNCTION LimitCheck_136 : BOOL
VAR_INPUT
    value : REAL;
    lo : REAL;
    hi : REAL;
END_VAR
    LimitCheck_136 := (value >= lo) AND (value <= hi);
END_FUNCTION

(* @LOOP_MAX(100) - 校验函数 137 *)
FUNCTION Verify_Channel_137 : INT
VAR_INPUT
    value : REAL;
    limit : REAL;
END_VAR
    tmp_bool := (value <= limit);
    IF tmp_bool THEN
        Verify_Channel_137 := 0;
    ELSE
        Verify_Channel_137 := -1;
    END_IF;
END_FUNCTION

FUNCTION Scale_137 : REAL
VAR_INPUT
    raw : REAL;
END_VAR
    tmp_real := raw * 1.137;
    IF tmp_real > 10000.0 THEN
        tmp_real := 10000.0;
    END_IF;
    Scale_137 := tmp_real;
END_FUNCTION

FUNCTION LimitCheck_137 : BOOL
VAR_INPUT
    value : REAL;
    lo : REAL;
    hi : REAL;
END_VAR
    LimitCheck_137 := (value >= lo) AND (value <= hi);
END_FUNCTION

(* @LOOP_MAX(100) - 校验函数 138 *)
FUNCTION Verify_Channel_138 : INT
VAR_INPUT
    value : REAL;
    limit : REAL;
END_VAR
    tmp_bool := (value <= limit);
    IF tmp_bool THEN
        Verify_Channel_138 := 0;
    ELSE
        Verify_Channel_138 := -1;
    END_IF;
END_FUNCTION

FUNCTION Scale_138 : REAL
VAR_INPUT
    raw : REAL;
END_VAR
    tmp_real := raw * 1.138;
    IF tmp_real > 10000.0 THEN
        tmp_real := 10000.0;
    END_IF;
    Scale_138 := tmp_real;
END_FUNCTION

FUNCTION LimitCheck_138 : BOOL
VAR_INPUT
    value : REAL;
    lo : REAL;
    hi : REAL;
END_VAR
    LimitCheck_138 := (value >= lo) AND (value <= hi);
END_FUNCTION

(* @LOOP_MAX(100) - 校验函数 139 *)
FUNCTION Verify_Channel_139 : INT
VAR_INPUT
    value : REAL;
    limit : REAL;
END_VAR
    tmp_bool := (value <= limit);
    IF tmp_bool THEN
        Verify_Channel_139 := 0;
    ELSE
        Verify_Channel_139 := -1;
    END_IF;
END_FUNCTION

FUNCTION Scale_139 : REAL
VAR_INPUT
    raw : REAL;
END_VAR
    tmp_real := raw * 1.139;
    IF tmp_real > 10000.0 THEN
        tmp_real := 10000.0;
    END_IF;
    Scale_139 := tmp_real;
END_FUNCTION

FUNCTION LimitCheck_139 : BOOL
VAR_INPUT
    value : REAL;
    lo : REAL;
    hi : REAL;
END_VAR
    LimitCheck_139 := (value >= lo) AND (value <= hi);
END_FUNCTION

(* @LOOP_MAX(100) - 校验函数 140 *)
FUNCTION Verify_Channel_140 : INT
VAR_INPUT
    value : REAL;
    limit : REAL;
END_VAR
    tmp_bool := (value <= limit);
    IF tmp_bool THEN
        Verify_Channel_140 := 0;
    ELSE
        Verify_Channel_140 := -1;
    END_IF;
END_FUNCTION

FUNCTION Scale_140 : REAL
VAR_INPUT
    raw : REAL;
END_VAR
    tmp_real := raw * 1.140;
    IF tmp_real > 10000.0 THEN
        tmp_real := 10000.0;
    END_IF;
    Scale_140 := tmp_real;
END_FUNCTION

FUNCTION LimitCheck_140 : BOOL
VAR_INPUT
    value : REAL;
    lo : REAL;
    hi : REAL;
END_VAR
    LimitCheck_140 := (value >= lo) AND (value <= hi);
END_FUNCTION

(* @LOOP_MAX(100) - 校验函数 141 *)
FUNCTION Verify_Channel_141 : INT
VAR_INPUT
    value : REAL;
    limit : REAL;
END_VAR
    tmp_bool := (value <= limit);
    IF tmp_bool THEN
        Verify_Channel_141 := 0;
    ELSE
        Verify_Channel_141 := -1;
    END_IF;
END_FUNCTION

FUNCTION Scale_141 : REAL
VAR_INPUT
    raw : REAL;
END_VAR
    tmp_real := raw * 1.141;
    IF tmp_real > 10000.0 THEN
        tmp_real := 10000.0;
    END_IF;
    Scale_141 := tmp_real;
END_FUNCTION

FUNCTION LimitCheck_141 : BOOL
VAR_INPUT
    value : REAL;
    lo : REAL;
    hi : REAL;
END_VAR
    LimitCheck_141 := (value >= lo) AND (value <= hi);
END_FUNCTION

(* @LOOP_MAX(100) - 校验函数 142 *)
FUNCTION Verify_Channel_142 : INT
VAR_INPUT
    value : REAL;
    limit : REAL;
END_VAR
    tmp_bool := (value <= limit);
    IF tmp_bool THEN
        Verify_Channel_142 := 0;
    ELSE
        Verify_Channel_142 := -1;
    END_IF;
END_FUNCTION

FUNCTION Scale_142 : REAL
VAR_INPUT
    raw : REAL;
END_VAR
    tmp_real := raw * 1.142;
    IF tmp_real > 10000.0 THEN
        tmp_real := 10000.0;
    END_IF;
    Scale_142 := tmp_real;
END_FUNCTION

FUNCTION LimitCheck_142 : BOOL
VAR_INPUT
    value : REAL;
    lo : REAL;
    hi : REAL;
END_VAR
    LimitCheck_142 := (value >= lo) AND (value <= hi);
END_FUNCTION

(* @LOOP_MAX(100) - 校验函数 143 *)
FUNCTION Verify_Channel_143 : INT
VAR_INPUT
    value : REAL;
    limit : REAL;
END_VAR
    tmp_bool := (value <= limit);
    IF tmp_bool THEN
        Verify_Channel_143 := 0;
    ELSE
        Verify_Channel_143 := -1;
    END_IF;
END_FUNCTION

FUNCTION Scale_143 : REAL
VAR_INPUT
    raw : REAL;
END_VAR
    tmp_real := raw * 1.143;
    IF tmp_real > 10000.0 THEN
        tmp_real := 10000.0;
    END_IF;
    Scale_143 := tmp_real;
END_FUNCTION

FUNCTION LimitCheck_143 : BOOL
VAR_INPUT
    value : REAL;
    lo : REAL;
    hi : REAL;
END_VAR
    LimitCheck_143 := (value >= lo) AND (value <= hi);
END_FUNCTION

(* @LOOP_MAX(100) - 校验函数 144 *)
FUNCTION Verify_Channel_144 : INT
VAR_INPUT
    value : REAL;
    limit : REAL;
END_VAR
    tmp_bool := (value <= limit);
    IF tmp_bool THEN
        Verify_Channel_144 := 0;
    ELSE
        Verify_Channel_144 := -1;
    END_IF;
END_FUNCTION

FUNCTION Scale_144 : REAL
VAR_INPUT
    raw : REAL;
END_VAR
    tmp_real := raw * 1.144;
    IF tmp_real > 10000.0 THEN
        tmp_real := 10000.0;
    END_IF;
    Scale_144 := tmp_real;
END_FUNCTION

FUNCTION LimitCheck_144 : BOOL
VAR_INPUT
    value : REAL;
    lo : REAL;
    hi : REAL;
END_VAR
    LimitCheck_144 := (value >= lo) AND (value <= hi);
END_FUNCTION

(* @LOOP_MAX(100) - 校验函数 145 *)
FUNCTION Verify_Channel_145 : INT
VAR_INPUT
    value : REAL;
    limit : REAL;
END_VAR
    tmp_bool := (value <= limit);
    IF tmp_bool THEN
        Verify_Channel_145 := 0;
    ELSE
        Verify_Channel_145 := -1;
    END_IF;
END_FUNCTION

FUNCTION Scale_145 : REAL
VAR_INPUT
    raw : REAL;
END_VAR
    tmp_real := raw * 1.145;
    IF tmp_real > 10000.0 THEN
        tmp_real := 10000.0;
    END_IF;
    Scale_145 := tmp_real;
END_FUNCTION

FUNCTION LimitCheck_145 : BOOL
VAR_INPUT
    value : REAL;
    lo : REAL;
    hi : REAL;
END_VAR
    LimitCheck_145 := (value >= lo) AND (value <= hi);
END_FUNCTION

(* @LOOP_MAX(100) - 校验函数 146 *)
FUNCTION Verify_Channel_146 : INT
VAR_INPUT
    value : REAL;
    limit : REAL;
END_VAR
    tmp_bool := (value <= limit);
    IF tmp_bool THEN
        Verify_Channel_146 := 0;
    ELSE
        Verify_Channel_146 := -1;
    END_IF;
END_FUNCTION

FUNCTION Scale_146 : REAL
VAR_INPUT
    raw : REAL;
END_VAR
    tmp_real := raw * 1.146;
    IF tmp_real > 10000.0 THEN
        tmp_real := 10000.0;
    END_IF;
    Scale_146 := tmp_real;
END_FUNCTION

FUNCTION LimitCheck_146 : BOOL
VAR_INPUT
    value : REAL;
    lo : REAL;
    hi : REAL;
END_VAR
    LimitCheck_146 := (value >= lo) AND (value <= hi);
END_FUNCTION

(* @LOOP_MAX(100) - 校验函数 147 *)
FUNCTION Verify_Channel_147 : INT
VAR_INPUT
    value : REAL;
    limit : REAL;
END_VAR
    tmp_bool := (value <= limit);
    IF tmp_bool THEN
        Verify_Channel_147 := 0;
    ELSE
        Verify_Channel_147 := -1;
    END_IF;
END_FUNCTION

FUNCTION Scale_147 : REAL
VAR_INPUT
    raw : REAL;
END_VAR
    tmp_real := raw * 1.147;
    IF tmp_real > 10000.0 THEN
        tmp_real := 10000.0;
    END_IF;
    Scale_147 := tmp_real;
END_FUNCTION

FUNCTION LimitCheck_147 : BOOL
VAR_INPUT
    value : REAL;
    lo : REAL;
    hi : REAL;
END_VAR
    LimitCheck_147 := (value >= lo) AND (value <= hi);
END_FUNCTION

(* @LOOP_MAX(100) - 校验函数 148 *)
FUNCTION Verify_Channel_148 : INT
VAR_INPUT
    value : REAL;
    limit : REAL;
END_VAR
    tmp_bool := (value <= limit);
    IF tmp_bool THEN
        Verify_Channel_148 := 0;
    ELSE
        Verify_Channel_148 := -1;
    END_IF;
END_FUNCTION

FUNCTION Scale_148 : REAL
VAR_INPUT
    raw : REAL;
END_VAR
    tmp_real := raw * 1.148;
    IF tmp_real > 10000.0 THEN
        tmp_real := 10000.0;
    END_IF;
    Scale_148 := tmp_real;
END_FUNCTION

FUNCTION LimitCheck_148 : BOOL
VAR_INPUT
    value : REAL;
    lo : REAL;
    hi : REAL;
END_VAR
    LimitCheck_148 := (value >= lo) AND (value <= hi);
END_FUNCTION

(* @LOOP_MAX(100) - 校验函数 149 *)
FUNCTION Verify_Channel_149 : INT
VAR_INPUT
    value : REAL;
    limit : REAL;
END_VAR
    tmp_bool := (value <= limit);
    IF tmp_bool THEN
        Verify_Channel_149 := 0;
    ELSE
        Verify_Channel_149 := -1;
    END_IF;
END_FUNCTION

FUNCTION Scale_149 : REAL
VAR_INPUT
    raw : REAL;
END_VAR
    tmp_real := raw * 1.149;
    IF tmp_real > 10000.0 THEN
        tmp_real := 10000.0;
    END_IF;
    Scale_149 := tmp_real;
END_FUNCTION

FUNCTION LimitCheck_149 : BOOL
VAR_INPUT
    value : REAL;
    lo : REAL;
    hi : REAL;
END_VAR
    LimitCheck_149 := (value >= lo) AND (value <= hi);
END_FUNCTION

(* @LOOP_MAX(100) - 校验函数 150 *)
FUNCTION Verify_Channel_150 : INT
VAR_INPUT
    value : REAL;
    limit : REAL;
END_VAR
    tmp_bool := (value <= limit);
    IF tmp_bool THEN
        Verify_Channel_150 := 0;
    ELSE
        Verify_Channel_150 := -1;
    END_IF;
END_FUNCTION

FUNCTION Scale_150 : REAL
VAR_INPUT
    raw : REAL;
END_VAR
    tmp_real := raw * 1.150;
    IF tmp_real > 10000.0 THEN
        tmp_real := 10000.0;
    END_IF;
    Scale_150 := tmp_real;
END_FUNCTION

FUNCTION LimitCheck_150 : BOOL
VAR_INPUT
    value : REAL;
    lo : REAL;
    hi : REAL;
END_VAR
    LimitCheck_150 := (value >= lo) AND (value <= hi);
END_FUNCTION

(* @LOOP_MAX(100) - 校验函数 151 *)
FUNCTION Verify_Channel_151 : INT
VAR_INPUT
    value : REAL;
    limit : REAL;
END_VAR
    tmp_bool := (value <= limit);
    IF tmp_bool THEN
        Verify_Channel_151 := 0;
    ELSE
        Verify_Channel_151 := -1;
    END_IF;
END_FUNCTION

FUNCTION Scale_151 : REAL
VAR_INPUT
    raw : REAL;
END_VAR
    tmp_real := raw * 1.151;
    IF tmp_real > 10000.0 THEN
        tmp_real := 10000.0;
    END_IF;
    Scale_151 := tmp_real;
END_FUNCTION

FUNCTION LimitCheck_151 : BOOL
VAR_INPUT
    value : REAL;
    lo : REAL;
    hi : REAL;
END_VAR
    LimitCheck_151 := (value >= lo) AND (value <= hi);
END_FUNCTION

(* @LOOP_MAX(100) - 校验函数 152 *)
FUNCTION Verify_Channel_152 : INT
VAR_INPUT
    value : REAL;
    limit : REAL;
END_VAR
    tmp_bool := (value <= limit);
    IF tmp_bool THEN
        Verify_Channel_152 := 0;
    ELSE
        Verify_Channel_152 := -1;
    END_IF;
END_FUNCTION

FUNCTION Scale_152 : REAL
VAR_INPUT
    raw : REAL;
END_VAR
    tmp_real := raw * 1.152;
    IF tmp_real > 10000.0 THEN
        tmp_real := 10000.0;
    END_IF;
    Scale_152 := tmp_real;
END_FUNCTION

FUNCTION LimitCheck_152 : BOOL
VAR_INPUT
    value : REAL;
    lo : REAL;
    hi : REAL;
END_VAR
    LimitCheck_152 := (value >= lo) AND (value <= hi);
END_FUNCTION

(* @LOOP_MAX(100) - 校验函数 153 *)
FUNCTION Verify_Channel_153 : INT
VAR_INPUT
    value : REAL;
    limit : REAL;
END_VAR
    tmp_bool := (value <= limit);
    IF tmp_bool THEN
        Verify_Channel_153 := 0;
    ELSE
        Verify_Channel_153 := -1;
    END_IF;
END_FUNCTION

FUNCTION Scale_153 : REAL
VAR_INPUT
    raw : REAL;
END_VAR
    tmp_real := raw * 1.153;
    IF tmp_real > 10000.0 THEN
        tmp_real := 10000.0;
    END_IF;
    Scale_153 := tmp_real;
END_FUNCTION

FUNCTION LimitCheck_153 : BOOL
VAR_INPUT
    value : REAL;
    lo : REAL;
    hi : REAL;
END_VAR
    LimitCheck_153 := (value >= lo) AND (value <= hi);
END_FUNCTION

(* @LOOP_MAX(100) - 校验函数 154 *)
FUNCTION Verify_Channel_154 : INT
VAR_INPUT
    value : REAL;
    limit : REAL;
END_VAR
    tmp_bool := (value <= limit);
    IF tmp_bool THEN
        Verify_Channel_154 := 0;
    ELSE
        Verify_Channel_154 := -1;
    END_IF;
END_FUNCTION

FUNCTION Scale_154 : REAL
VAR_INPUT
    raw : REAL;
END_VAR
    tmp_real := raw * 1.154;
    IF tmp_real > 10000.0 THEN
        tmp_real := 10000.0;
    END_IF;
    Scale_154 := tmp_real;
END_FUNCTION

FUNCTION LimitCheck_154 : BOOL
VAR_INPUT
    value : REAL;
    lo : REAL;
    hi : REAL;
END_VAR
    LimitCheck_154 := (value >= lo) AND (value <= hi);
END_FUNCTION

(* @LOOP_MAX(100) - 校验函数 155 *)
FUNCTION Verify_Channel_155 : INT
VAR_INPUT
    value : REAL;
    limit : REAL;
END_VAR
    tmp_bool := (value <= limit);
    IF tmp_bool THEN
        Verify_Channel_155 := 0;
    ELSE
        Verify_Channel_155 := -1;
    END_IF;
END_FUNCTION

FUNCTION Scale_155 : REAL
VAR_INPUT
    raw : REAL;
END_VAR
    tmp_real := raw * 1.155;
    IF tmp_real > 10000.0 THEN
        tmp_real := 10000.0;
    END_IF;
    Scale_155 := tmp_real;
END_FUNCTION

FUNCTION LimitCheck_155 : BOOL
VAR_INPUT
    value : REAL;
    lo : REAL;
    hi : REAL;
END_VAR
    LimitCheck_155 := (value >= lo) AND (value <= hi);
END_FUNCTION

(* @LOOP_MAX(100) - 校验函数 156 *)
FUNCTION Verify_Channel_156 : INT
VAR_INPUT
    value : REAL;
    limit : REAL;
END_VAR
    tmp_bool := (value <= limit);
    IF tmp_bool THEN
        Verify_Channel_156 := 0;
    ELSE
        Verify_Channel_156 := -1;
    END_IF;
END_FUNCTION

FUNCTION Scale_156 : REAL
VAR_INPUT
    raw : REAL;
END_VAR
    tmp_real := raw * 1.156;
    IF tmp_real > 10000.0 THEN
        tmp_real := 10000.0;
    END_IF;
    Scale_156 := tmp_real;
END_FUNCTION

FUNCTION LimitCheck_156 : BOOL
VAR_INPUT
    value : REAL;
    lo : REAL;
    hi : REAL;
END_VAR
    LimitCheck_156 := (value >= lo) AND (value <= hi);
END_FUNCTION

(* @LOOP_MAX(100) - 校验函数 157 *)
FUNCTION Verify_Channel_157 : INT
VAR_INPUT
    value : REAL;
    limit : REAL;
END_VAR
    tmp_bool := (value <= limit);
    IF tmp_bool THEN
        Verify_Channel_157 := 0;
    ELSE
        Verify_Channel_157 := -1;
    END_IF;
END_FUNCTION

FUNCTION Scale_157 : REAL
VAR_INPUT
    raw : REAL;
END_VAR
    tmp_real := raw * 1.157;
    IF tmp_real > 10000.0 THEN
        tmp_real := 10000.0;
    END_IF;
    Scale_157 := tmp_real;
END_FUNCTION

FUNCTION LimitCheck_157 : BOOL
VAR_INPUT
    value : REAL;
    lo : REAL;
    hi : REAL;
END_VAR
    LimitCheck_157 := (value >= lo) AND (value <= hi);
END_FUNCTION

(* @LOOP_MAX(100) - 校验函数 158 *)
FUNCTION Verify_Channel_158 : INT
VAR_INPUT
    value : REAL;
    limit : REAL;
END_VAR
    tmp_bool := (value <= limit);
    IF tmp_bool THEN
        Verify_Channel_158 := 0;
    ELSE
        Verify_Channel_158 := -1;
    END_IF;
END_FUNCTION

FUNCTION Scale_158 : REAL
VAR_INPUT
    raw : REAL;
END_VAR
    tmp_real := raw * 1.158;
    IF tmp_real > 10000.0 THEN
        tmp_real := 10000.0;
    END_IF;
    Scale_158 := tmp_real;
END_FUNCTION

FUNCTION LimitCheck_158 : BOOL
VAR_INPUT
    value : REAL;
    lo : REAL;
    hi : REAL;
END_VAR
    LimitCheck_158 := (value >= lo) AND (value <= hi);
END_FUNCTION

(* @LOOP_MAX(100) - 校验函数 159 *)
FUNCTION Verify_Channel_159 : INT
VAR_INPUT
    value : REAL;
    limit : REAL;
END_VAR
    tmp_bool := (value <= limit);
    IF tmp_bool THEN
        Verify_Channel_159 := 0;
    ELSE
        Verify_Channel_159 := -1;
    END_IF;
END_FUNCTION

FUNCTION Scale_159 : REAL
VAR_INPUT
    raw : REAL;
END_VAR
    tmp_real := raw * 1.159;
    IF tmp_real > 10000.0 THEN
        tmp_real := 10000.0;
    END_IF;
    Scale_159 := tmp_real;
END_FUNCTION

FUNCTION LimitCheck_159 : BOOL
VAR_INPUT
    value : REAL;
    lo : REAL;
    hi : REAL;
END_VAR
    LimitCheck_159 := (value >= lo) AND (value <= hi);
END_FUNCTION

(* @LOOP_MAX(100) - 校验函数 160 *)
FUNCTION Verify_Channel_160 : INT
VAR_INPUT
    value : REAL;
    limit : REAL;
END_VAR
    tmp_bool := (value <= limit);
    IF tmp_bool THEN
        Verify_Channel_160 := 0;
    ELSE
        Verify_Channel_160 := -1;
    END_IF;
END_FUNCTION

FUNCTION Scale_160 : REAL
VAR_INPUT
    raw : REAL;
END_VAR
    tmp_real := raw * 1.160;
    IF tmp_real > 10000.0 THEN
        tmp_real := 10000.0;
    END_IF;
    Scale_160 := tmp_real;
END_FUNCTION

FUNCTION LimitCheck_160 : BOOL
VAR_INPUT
    value : REAL;
    lo : REAL;
    hi : REAL;
END_VAR
    LimitCheck_160 := (value >= lo) AND (value <= hi);
END_FUNCTION

(* @LOOP_MAX(100) - 校验函数 161 *)
FUNCTION Verify_Channel_161 : INT
VAR_INPUT
    value : REAL;
    limit : REAL;
END_VAR
    tmp_bool := (value <= limit);
    IF tmp_bool THEN
        Verify_Channel_161 := 0;
    ELSE
        Verify_Channel_161 := -1;
    END_IF;
END_FUNCTION

FUNCTION Scale_161 : REAL
VAR_INPUT
    raw : REAL;
END_VAR
    tmp_real := raw * 1.161;
    IF tmp_real > 10000.0 THEN
        tmp_real := 10000.0;
    END_IF;
    Scale_161 := tmp_real;
END_FUNCTION

FUNCTION LimitCheck_161 : BOOL
VAR_INPUT
    value : REAL;
    lo : REAL;
    hi : REAL;
END_VAR
    LimitCheck_161 := (value >= lo) AND (value <= hi);
END_FUNCTION

(* @LOOP_MAX(100) - 校验函数 162 *)
FUNCTION Verify_Channel_162 : INT
VAR_INPUT
    value : REAL;
    limit : REAL;
END_VAR
    tmp_bool := (value <= limit);
    IF tmp_bool THEN
        Verify_Channel_162 := 0;
    ELSE
        Verify_Channel_162 := -1;
    END_IF;
END_FUNCTION

FUNCTION Scale_162 : REAL
VAR_INPUT
    raw : REAL;
END_VAR
    tmp_real := raw * 1.162;
    IF tmp_real > 10000.0 THEN
        tmp_real := 10000.0;
    END_IF;
    Scale_162 := tmp_real;
END_FUNCTION

FUNCTION LimitCheck_162 : BOOL
VAR_INPUT
    value : REAL;
    lo : REAL;
    hi : REAL;
END_VAR
    LimitCheck_162 := (value >= lo) AND (value <= hi);
END_FUNCTION

(* @LOOP_MAX(100) - 校验函数 163 *)
FUNCTION Verify_Channel_163 : INT
VAR_INPUT
    value : REAL;
    limit : REAL;
END_VAR
    tmp_bool := (value <= limit);
    IF tmp_bool THEN
        Verify_Channel_163 := 0;
    ELSE
        Verify_Channel_163 := -1;
    END_IF;
END_FUNCTION

FUNCTION Scale_163 : REAL
VAR_INPUT
    raw : REAL;
END_VAR
    tmp_real := raw * 1.163;
    IF tmp_real > 10000.0 THEN
        tmp_real := 10000.0;
    END_IF;
    Scale_163 := tmp_real;
END_FUNCTION

FUNCTION LimitCheck_163 : BOOL
VAR_INPUT
    value : REAL;
    lo : REAL;
    hi : REAL;
END_VAR
    LimitCheck_163 := (value >= lo) AND (value <= hi);
END_FUNCTION

(* @LOOP_MAX(100) - 校验函数 164 *)
FUNCTION Verify_Channel_164 : INT
VAR_INPUT
    value : REAL;
    limit : REAL;
END_VAR
    tmp_bool := (value <= limit);
    IF tmp_bool THEN
        Verify_Channel_164 := 0;
    ELSE
        Verify_Channel_164 := -1;
    END_IF;
END_FUNCTION

FUNCTION Scale_164 : REAL
VAR_INPUT
    raw : REAL;
END_VAR
    tmp_real := raw * 1.164;
    IF tmp_real > 10000.0 THEN
        tmp_real := 10000.0;
    END_IF;
    Scale_164 := tmp_real;
END_FUNCTION

FUNCTION LimitCheck_164 : BOOL
VAR_INPUT
    value : REAL;
    lo : REAL;
    hi : REAL;
END_VAR
    LimitCheck_164 := (value >= lo) AND (value <= hi);
END_FUNCTION

(* @LOOP_MAX(100) - 校验函数 165 *)
FUNCTION Verify_Channel_165 : INT
VAR_INPUT
    value : REAL;
    limit : REAL;
END_VAR
    tmp_bool := (value <= limit);
    IF tmp_bool THEN
        Verify_Channel_165 := 0;
    ELSE
        Verify_Channel_165 := -1;
    END_IF;
END_FUNCTION

FUNCTION Scale_165 : REAL
VAR_INPUT
    raw : REAL;
END_VAR
    tmp_real := raw * 1.165;
    IF tmp_real > 10000.0 THEN
        tmp_real := 10000.0;
    END_IF;
    Scale_165 := tmp_real;
END_FUNCTION

FUNCTION LimitCheck_165 : BOOL
VAR_INPUT
    value : REAL;
    lo : REAL;
    hi : REAL;
END_VAR
    LimitCheck_165 := (value >= lo) AND (value <= hi);
END_FUNCTION

(* @LOOP_MAX(100) - 校验函数 166 *)
FUNCTION Verify_Channel_166 : INT
VAR_INPUT
    value : REAL;
    limit : REAL;
END_VAR
    tmp_bool := (value <= limit);
    IF tmp_bool THEN
        Verify_Channel_166 := 0;
    ELSE
        Verify_Channel_166 := -1;
    END_IF;
END_FUNCTION

FUNCTION Scale_166 : REAL
VAR_INPUT
    raw : REAL;
END_VAR
    tmp_real := raw * 1.166;
    IF tmp_real > 10000.0 THEN
        tmp_real := 10000.0;
    END_IF;
    Scale_166 := tmp_real;
END_FUNCTION

FUNCTION LimitCheck_166 : BOOL
VAR_INPUT
    value : REAL;
    lo : REAL;
    hi : REAL;
END_VAR
    LimitCheck_166 := (value >= lo) AND (value <= hi);
END_FUNCTION

(* @LOOP_MAX(100) - 校验函数 167 *)
FUNCTION Verify_Channel_167 : INT
VAR_INPUT
    value : REAL;
    limit : REAL;
END_VAR
    tmp_bool := (value <= limit);
    IF tmp_bool THEN
        Verify_Channel_167 := 0;
    ELSE
        Verify_Channel_167 := -1;
    END_IF;
END_FUNCTION

FUNCTION Scale_167 : REAL
VAR_INPUT
    raw : REAL;
END_VAR
    tmp_real := raw * 1.167;
    IF tmp_real > 10000.0 THEN
        tmp_real := 10000.0;
    END_IF;
    Scale_167 := tmp_real;
END_FUNCTION

FUNCTION LimitCheck_167 : BOOL
VAR_INPUT
    value : REAL;
    lo : REAL;
    hi : REAL;
END_VAR
    LimitCheck_167 := (value >= lo) AND (value <= hi);
END_FUNCTION

(* @LOOP_MAX(100) - 校验函数 168 *)
FUNCTION Verify_Channel_168 : INT
VAR_INPUT
    value : REAL;
    limit : REAL;
END_VAR
    tmp_bool := (value <= limit);
    IF tmp_bool THEN
        Verify_Channel_168 := 0;
    ELSE
        Verify_Channel_168 := -1;
    END_IF;
END_FUNCTION

FUNCTION Scale_168 : REAL
VAR_INPUT
    raw : REAL;
END_VAR
    tmp_real := raw * 1.168;
    IF tmp_real > 10000.0 THEN
        tmp_real := 10000.0;
    END_IF;
    Scale_168 := tmp_real;
END_FUNCTION

FUNCTION LimitCheck_168 : BOOL
VAR_INPUT
    value : REAL;
    lo : REAL;
    hi : REAL;
END_VAR
    LimitCheck_168 := (value >= lo) AND (value <= hi);
END_FUNCTION

(* @LOOP_MAX(100) - 校验函数 169 *)
FUNCTION Verify_Channel_169 : INT
VAR_INPUT
    value : REAL;
    limit : REAL;
END_VAR
    tmp_bool := (value <= limit);
    IF tmp_bool THEN
        Verify_Channel_169 := 0;
    ELSE
        Verify_Channel_169 := -1;
    END_IF;
END_FUNCTION

FUNCTION Scale_169 : REAL
VAR_INPUT
    raw : REAL;
END_VAR
    tmp_real := raw * 1.169;
    IF tmp_real > 10000.0 THEN
        tmp_real := 10000.0;
    END_IF;
    Scale_169 := tmp_real;
END_FUNCTION

FUNCTION LimitCheck_169 : BOOL
VAR_INPUT
    value : REAL;
    lo : REAL;
    hi : REAL;
END_VAR
    LimitCheck_169 := (value >= lo) AND (value <= hi);
END_FUNCTION

(* @LOOP_MAX(100) - 校验函数 170 *)
FUNCTION Verify_Channel_170 : INT
VAR_INPUT
    value : REAL;
    limit : REAL;
END_VAR
    tmp_bool := (value <= limit);
    IF tmp_bool THEN
        Verify_Channel_170 := 0;
    ELSE
        Verify_Channel_170 := -1;
    END_IF;
END_FUNCTION

FUNCTION Scale_170 : REAL
VAR_INPUT
    raw : REAL;
END_VAR
    tmp_real := raw * 1.170;
    IF tmp_real > 10000.0 THEN
        tmp_real := 10000.0;
    END_IF;
    Scale_170 := tmp_real;
END_FUNCTION

FUNCTION LimitCheck_170 : BOOL
VAR_INPUT
    value : REAL;
    lo : REAL;
    hi : REAL;
END_VAR
    LimitCheck_170 := (value >= lo) AND (value <= hi);
END_FUNCTION

(* @LOOP_MAX(100) - 校验函数 171 *)
FUNCTION Verify_Channel_171 : INT
VAR_INPUT
    value : REAL;
    limit : REAL;
END_VAR
    tmp_bool := (value <= limit);
    IF tmp_bool THEN
        Verify_Channel_171 := 0;
    ELSE
        Verify_Channel_171 := -1;
    END_IF;
END_FUNCTION

FUNCTION Scale_171 : REAL
VAR_INPUT
    raw : REAL;
END_VAR
    tmp_real := raw * 1.171;
    IF tmp_real > 10000.0 THEN
        tmp_real := 10000.0;
    END_IF;
    Scale_171 := tmp_real;
END_FUNCTION

FUNCTION LimitCheck_171 : BOOL
VAR_INPUT
    value : REAL;
    lo : REAL;
    hi : REAL;
END_VAR
    LimitCheck_171 := (value >= lo) AND (value <= hi);
END_FUNCTION

(* @LOOP_MAX(100) - 校验函数 172 *)
FUNCTION Verify_Channel_172 : INT
VAR_INPUT
    value : REAL;
    limit : REAL;
END_VAR
    tmp_bool := (value <= limit);
    IF tmp_bool THEN
        Verify_Channel_172 := 0;
    ELSE
        Verify_Channel_172 := -1;
    END_IF;
END_FUNCTION

FUNCTION Scale_172 : REAL
VAR_INPUT
    raw : REAL;
END_VAR
    tmp_real := raw * 1.172;
    IF tmp_real > 10000.0 THEN
        tmp_real := 10000.0;
    END_IF;
    Scale_172 := tmp_real;
END_FUNCTION

FUNCTION LimitCheck_172 : BOOL
VAR_INPUT
    value : REAL;
    lo : REAL;
    hi : REAL;
END_VAR
    LimitCheck_172 := (value >= lo) AND (value <= hi);
END_FUNCTION

(* @LOOP_MAX(100) - 校验函数 173 *)
FUNCTION Verify_Channel_173 : INT
VAR_INPUT
    value : REAL;
    limit : REAL;
END_VAR
    tmp_bool := (value <= limit);
    IF tmp_bool THEN
        Verify_Channel_173 := 0;
    ELSE
        Verify_Channel_173 := -1;
    END_IF;
END_FUNCTION

FUNCTION Scale_173 : REAL
VAR_INPUT
    raw : REAL;
END_VAR
    tmp_real := raw * 1.173;
    IF tmp_real > 10000.0 THEN
        tmp_real := 10000.0;
    END_IF;
    Scale_173 := tmp_real;
END_FUNCTION

FUNCTION LimitCheck_173 : BOOL
VAR_INPUT
    value : REAL;
    lo : REAL;
    hi : REAL;
END_VAR
    LimitCheck_173 := (value >= lo) AND (value <= hi);
END_FUNCTION

(* @LOOP_MAX(100) - 校验函数 174 *)
FUNCTION Verify_Channel_174 : INT
VAR_INPUT
    value : REAL;
    limit : REAL;
END_VAR
    tmp_bool := (value <= limit);
    IF tmp_bool THEN
        Verify_Channel_174 := 0;
    ELSE
        Verify_Channel_174 := -1;
    END_IF;
END_FUNCTION

FUNCTION Scale_174 : REAL
VAR_INPUT
    raw : REAL;
END_VAR
    tmp_real := raw * 1.174;
    IF tmp_real > 10000.0 THEN
        tmp_real := 10000.0;
    END_IF;
    Scale_174 := tmp_real;
END_FUNCTION

FUNCTION LimitCheck_174 : BOOL
VAR_INPUT
    value : REAL;
    lo : REAL;
    hi : REAL;
END_VAR
    LimitCheck_174 := (value >= lo) AND (value <= hi);
END_FUNCTION

(* @LOOP_MAX(100) - 校验函数 175 *)
FUNCTION Verify_Channel_175 : INT
VAR_INPUT
    value : REAL;
    limit : REAL;
END_VAR
    tmp_bool := (value <= limit);
    IF tmp_bool THEN
        Verify_Channel_175 := 0;
    ELSE
        Verify_Channel_175 := -1;
    END_IF;
END_FUNCTION

FUNCTION Scale_175 : REAL
VAR_INPUT
    raw : REAL;
END_VAR
    tmp_real := raw * 1.175;
    IF tmp_real > 10000.0 THEN
        tmp_real := 10000.0;
    END_IF;
    Scale_175 := tmp_real;
END_FUNCTION

FUNCTION LimitCheck_175 : BOOL
VAR_INPUT
    value : REAL;
    lo : REAL;
    hi : REAL;
END_VAR
    LimitCheck_175 := (value >= lo) AND (value <= hi);
END_FUNCTION

(* @LOOP_MAX(100) - 校验函数 176 *)
FUNCTION Verify_Channel_176 : INT
VAR_INPUT
    value : REAL;
    limit : REAL;
END_VAR
    tmp_bool := (value <= limit);
    IF tmp_bool THEN
        Verify_Channel_176 := 0;
    ELSE
        Verify_Channel_176 := -1;
    END_IF;
END_FUNCTION

FUNCTION Scale_176 : REAL
VAR_INPUT
    raw : REAL;
END_VAR
    tmp_real := raw * 1.176;
    IF tmp_real > 10000.0 THEN
        tmp_real := 10000.0;
    END_IF;
    Scale_176 := tmp_real;
END_FUNCTION

FUNCTION LimitCheck_176 : BOOL
VAR_INPUT
    value : REAL;
    lo : REAL;
    hi : REAL;
END_VAR
    LimitCheck_176 := (value >= lo) AND (value <= hi);
END_FUNCTION

(* @LOOP_MAX(100) - 校验函数 177 *)
FUNCTION Verify_Channel_177 : INT
VAR_INPUT
    value : REAL;
    limit : REAL;
END_VAR
    tmp_bool := (value <= limit);
    IF tmp_bool THEN
        Verify_Channel_177 := 0;
    ELSE
        Verify_Channel_177 := -1;
    END_IF;
END_FUNCTION

FUNCTION Scale_177 : REAL
VAR_INPUT
    raw : REAL;
END_VAR
    tmp_real := raw * 1.177;
    IF tmp_real > 10000.0 THEN
        tmp_real := 10000.0;
    END_IF;
    Scale_177 := tmp_real;
END_FUNCTION

FUNCTION LimitCheck_177 : BOOL
VAR_INPUT
    value : REAL;
    lo : REAL;
    hi : REAL;
END_VAR
    LimitCheck_177 := (value >= lo) AND (value <= hi);
END_FUNCTION

(* @LOOP_MAX(100) - 校验函数 178 *)
FUNCTION Verify_Channel_178 : INT
VAR_INPUT
    value : REAL;
    limit : REAL;
END_VAR
    tmp_bool := (value <= limit);
    IF tmp_bool THEN
        Verify_Channel_178 := 0;
    ELSE
        Verify_Channel_178 := -1;
    END_IF;
END_FUNCTION

FUNCTION Scale_178 : REAL
VAR_INPUT
    raw : REAL;
END_VAR
    tmp_real := raw * 1.178;
    IF tmp_real > 10000.0 THEN
        tmp_real := 10000.0;
    END_IF;
    Scale_178 := tmp_real;
END_FUNCTION

FUNCTION LimitCheck_178 : BOOL
VAR_INPUT
    value : REAL;
    lo : REAL;
    hi : REAL;
END_VAR
    LimitCheck_178 := (value >= lo) AND (value <= hi);
END_FUNCTION

(* @LOOP_MAX(100) - 校验函数 179 *)
FUNCTION Verify_Channel_179 : INT
VAR_INPUT
    value : REAL;
    limit : REAL;
END_VAR
    tmp_bool := (value <= limit);
    IF tmp_bool THEN
        Verify_Channel_179 := 0;
    ELSE
        Verify_Channel_179 := -1;
    END_IF;
END_FUNCTION

FUNCTION Scale_179 : REAL
VAR_INPUT
    raw : REAL;
END_VAR
    tmp_real := raw * 1.179;
    IF tmp_real > 10000.0 THEN
        tmp_real := 10000.0;
    END_IF;
    Scale_179 := tmp_real;
END_FUNCTION

FUNCTION LimitCheck_179 : BOOL
VAR_INPUT
    value : REAL;
    lo : REAL;
    hi : REAL;
END_VAR
    LimitCheck_179 := (value >= lo) AND (value <= hi);
END_FUNCTION

(* @LOOP_MAX(100) - 校验函数 180 *)
FUNCTION Verify_Channel_180 : INT
VAR_INPUT
    value : REAL;
    limit : REAL;
END_VAR
    tmp_bool := (value <= limit);
    IF tmp_bool THEN
        Verify_Channel_180 := 0;
    ELSE
        Verify_Channel_180 := -1;
    END_IF;
END_FUNCTION

FUNCTION Scale_180 : REAL
VAR_INPUT
    raw : REAL;
END_VAR
    tmp_real := raw * 1.180;
    IF tmp_real > 10000.0 THEN
        tmp_real := 10000.0;
    END_IF;
    Scale_180 := tmp_real;
END_FUNCTION

FUNCTION LimitCheck_180 : BOOL
VAR_INPUT
    value : REAL;
    lo : REAL;
    hi : REAL;
END_VAR
    LimitCheck_180 := (value >= lo) AND (value <= hi);
END_FUNCTION

(* @LOOP_MAX(100) - 校验函数 181 *)
FUNCTION Verify_Channel_181 : INT
VAR_INPUT
    value : REAL;
    limit : REAL;
END_VAR
    tmp_bool := (value <= limit);
    IF tmp_bool THEN
        Verify_Channel_181 := 0;
    ELSE
        Verify_Channel_181 := -1;
    END_IF;
END_FUNCTION

FUNCTION Scale_181 : REAL
VAR_INPUT
    raw : REAL;
END_VAR
    tmp_real := raw * 1.181;
    IF tmp_real > 10000.0 THEN
        tmp_real := 10000.0;
    END_IF;
    Scale_181 := tmp_real;
END_FUNCTION

FUNCTION LimitCheck_181 : BOOL
VAR_INPUT
    value : REAL;
    lo : REAL;
    hi : REAL;
END_VAR
    LimitCheck_181 := (value >= lo) AND (value <= hi);
END_FUNCTION

(* @LOOP_MAX(100) - 校验函数 182 *)
FUNCTION Verify_Channel_182 : INT
VAR_INPUT
    value : REAL;
    limit : REAL;
END_VAR
    tmp_bool := (value <= limit);
    IF tmp_bool THEN
        Verify_Channel_182 := 0;
    ELSE
        Verify_Channel_182 := -1;
    END_IF;
END_FUNCTION

FUNCTION Scale_182 : REAL
VAR_INPUT
    raw : REAL;
END_VAR
    tmp_real := raw * 1.182;
    IF tmp_real > 10000.0 THEN
        tmp_real := 10000.0;
    END_IF;
    Scale_182 := tmp_real;
END_FUNCTION

FUNCTION LimitCheck_182 : BOOL
VAR_INPUT
    value : REAL;
    lo : REAL;
    hi : REAL;
END_VAR
    LimitCheck_182 := (value >= lo) AND (value <= hi);
END_FUNCTION

(* @LOOP_MAX(100) - 校验函数 183 *)
FUNCTION Verify_Channel_183 : INT
VAR_INPUT
    value : REAL;
    limit : REAL;
END_VAR
    tmp_bool := (value <= limit);
    IF tmp_bool THEN
        Verify_Channel_183 := 0;
    ELSE
        Verify_Channel_183 := -1;
    END_IF;
END_FUNCTION

FUNCTION Scale_183 : REAL
VAR_INPUT
    raw : REAL;
END_VAR
    tmp_real := raw * 1.183;
    IF tmp_real > 10000.0 THEN
        tmp_real := 10000.0;
    END_IF;
    Scale_183 := tmp_real;
END_FUNCTION

FUNCTION LimitCheck_183 : BOOL
VAR_INPUT
    value : REAL;
    lo : REAL;
    hi : REAL;
END_VAR
    LimitCheck_183 := (value >= lo) AND (value <= hi);
END_FUNCTION

(* @LOOP_MAX(100) - 校验函数 184 *)
FUNCTION Verify_Channel_184 : INT
VAR_INPUT
    value : REAL;
    limit : REAL;
END_VAR
    tmp_bool := (value <= limit);
    IF tmp_bool THEN
        Verify_Channel_184 := 0;
    ELSE
        Verify_Channel_184 := -1;
    END_IF;
END_FUNCTION

FUNCTION Scale_184 : REAL
VAR_INPUT
    raw : REAL;
END_VAR
    tmp_real := raw * 1.184;
    IF tmp_real > 10000.0 THEN
        tmp_real := 10000.0;
    END_IF;
    Scale_184 := tmp_real;
END_FUNCTION

FUNCTION LimitCheck_184 : BOOL
VAR_INPUT
    value : REAL;
    lo : REAL;
    hi : REAL;
END_VAR
    LimitCheck_184 := (value >= lo) AND (value <= hi);
END_FUNCTION

(* @LOOP_MAX(100) - 校验函数 185 *)
FUNCTION Verify_Channel_185 : INT
VAR_INPUT
    value : REAL;
    limit : REAL;
END_VAR
    tmp_bool := (value <= limit);
    IF tmp_bool THEN
        Verify_Channel_185 := 0;
    ELSE
        Verify_Channel_185 := -1;
    END_IF;
END_FUNCTION

FUNCTION Scale_185 : REAL
VAR_INPUT
    raw : REAL;
END_VAR
    tmp_real := raw * 1.185;
    IF tmp_real > 10000.0 THEN
        tmp_real := 10000.0;
    END_IF;
    Scale_185 := tmp_real;
END_FUNCTION

FUNCTION LimitCheck_185 : BOOL
VAR_INPUT
    value : REAL;
    lo : REAL;
    hi : REAL;
END_VAR
    LimitCheck_185 := (value >= lo) AND (value <= hi);
END_FUNCTION

(* @LOOP_MAX(100) - 校验函数 186 *)
FUNCTION Verify_Channel_186 : INT
VAR_INPUT
    value : REAL;
    limit : REAL;
END_VAR
    tmp_bool := (value <= limit);
    IF tmp_bool THEN
        Verify_Channel_186 := 0;
    ELSE
        Verify_Channel_186 := -1;
    END_IF;
END_FUNCTION

FUNCTION Scale_186 : REAL
VAR_INPUT
    raw : REAL;
END_VAR
    tmp_real := raw * 1.186;
    IF tmp_real > 10000.0 THEN
        tmp_real := 10000.0;
    END_IF;
    Scale_186 := tmp_real;
END_FUNCTION

FUNCTION LimitCheck_186 : BOOL
VAR_INPUT
    value : REAL;
    lo : REAL;
    hi : REAL;
END_VAR
    LimitCheck_186 := (value >= lo) AND (value <= hi);
END_FUNCTION

(* @LOOP_MAX(100) - 校验函数 187 *)
FUNCTION Verify_Channel_187 : INT
VAR_INPUT
    value : REAL;
    limit : REAL;
END_VAR
    tmp_bool := (value <= limit);
    IF tmp_bool THEN
        Verify_Channel_187 := 0;
    ELSE
        Verify_Channel_187 := -1;
    END_IF;
END_FUNCTION

FUNCTION Scale_187 : REAL
VAR_INPUT
    raw : REAL;
END_VAR
    tmp_real := raw * 1.187;
    IF tmp_real > 10000.0 THEN
        tmp_real := 10000.0;
    END_IF;
    Scale_187 := tmp_real;
END_FUNCTION

FUNCTION LimitCheck_187 : BOOL
VAR_INPUT
    value : REAL;
    lo : REAL;
    hi : REAL;
END_VAR
    LimitCheck_187 := (value >= lo) AND (value <= hi);
END_FUNCTION

(* @LOOP_MAX(100) - 校验函数 188 *)
FUNCTION Verify_Channel_188 : INT
VAR_INPUT
    value : REAL;
    limit : REAL;
END_VAR
    tmp_bool := (value <= limit);
    IF tmp_bool THEN
        Verify_Channel_188 := 0;
    ELSE
        Verify_Channel_188 := -1;
    END_IF;
END_FUNCTION

FUNCTION Scale_188 : REAL
VAR_INPUT
    raw : REAL;
END_VAR
    tmp_real := raw * 1.188;
    IF tmp_real > 10000.0 THEN
        tmp_real := 10000.0;
    END_IF;
    Scale_188 := tmp_real;
END_FUNCTION

FUNCTION LimitCheck_188 : BOOL
VAR_INPUT
    value : REAL;
    lo : REAL;
    hi : REAL;
END_VAR
    LimitCheck_188 := (value >= lo) AND (value <= hi);
END_FUNCTION

(* @LOOP_MAX(100) - 校验函数 189 *)
FUNCTION Verify_Channel_189 : INT
VAR_INPUT
    value : REAL;
    limit : REAL;
END_VAR
    tmp_bool := (value <= limit);
    IF tmp_bool THEN
        Verify_Channel_189 := 0;
    ELSE
        Verify_Channel_189 := -1;
    END_IF;
END_FUNCTION

FUNCTION Scale_189 : REAL
VAR_INPUT
    raw : REAL;
END_VAR
    tmp_real := raw * 1.189;
    IF tmp_real > 10000.0 THEN
        tmp_real := 10000.0;
    END_IF;
    Scale_189 := tmp_real;
END_FUNCTION

FUNCTION LimitCheck_189 : BOOL
VAR_INPUT
    value : REAL;
    lo : REAL;
    hi : REAL;
END_VAR
    LimitCheck_189 := (value >= lo) AND (value <= hi);
END_FUNCTION

(* @LOOP_MAX(100) - 校验函数 190 *)
FUNCTION Verify_Channel_190 : INT
VAR_INPUT
    value : REAL;
    limit : REAL;
END_VAR
    tmp_bool := (value <= limit);
    IF tmp_bool THEN
        Verify_Channel_190 := 0;
    ELSE
        Verify_Channel_190 := -1;
    END_IF;
END_FUNCTION

FUNCTION Scale_190 : REAL
VAR_INPUT
    raw : REAL;
END_VAR
    tmp_real := raw * 1.190;
    IF tmp_real > 10000.0 THEN
        tmp_real := 10000.0;
    END_IF;
    Scale_190 := tmp_real;
END_FUNCTION

FUNCTION LimitCheck_190 : BOOL
VAR_INPUT
    value : REAL;
    lo : REAL;
    hi : REAL;
END_VAR
    LimitCheck_190 := (value >= lo) AND (value <= hi);
END_FUNCTION

(* @LOOP_MAX(100) - 校验函数 191 *)
FUNCTION Verify_Channel_191 : INT
VAR_INPUT
    value : REAL;
    limit : REAL;
END_VAR
    tmp_bool := (value <= limit);
    IF tmp_bool THEN
        Verify_Channel_191 := 0;
    ELSE
        Verify_Channel_191 := -1;
    END_IF;
END_FUNCTION

FUNCTION Scale_191 : REAL
VAR_INPUT
    raw : REAL;
END_VAR
    tmp_real := raw * 1.191;
    IF tmp_real > 10000.0 THEN
        tmp_real := 10000.0;
    END_IF;
    Scale_191 := tmp_real;
END_FUNCTION

FUNCTION LimitCheck_191 : BOOL
VAR_INPUT
    value : REAL;
    lo : REAL;
    hi : REAL;
END_VAR
    LimitCheck_191 := (value >= lo) AND (value <= hi);
END_FUNCTION

(* @LOOP_MAX(100) - 校验函数 192 *)
FUNCTION Verify_Channel_192 : INT
VAR_INPUT
    value : REAL;
    limit : REAL;
END_VAR
    tmp_bool := (value <= limit);
    IF tmp_bool THEN
        Verify_Channel_192 := 0;
    ELSE
        Verify_Channel_192 := -1;
    END_IF;
END_FUNCTION

FUNCTION Scale_192 : REAL
VAR_INPUT
    raw : REAL;
END_VAR
    tmp_real := raw * 1.192;
    IF tmp_real > 10000.0 THEN
        tmp_real := 10000.0;
    END_IF;
    Scale_192 := tmp_real;
END_FUNCTION

FUNCTION LimitCheck_192 : BOOL
VAR_INPUT
    value : REAL;
    lo : REAL;
    hi : REAL;
END_VAR
    LimitCheck_192 := (value >= lo) AND (value <= hi);
END_FUNCTION

(* @LOOP_MAX(100) - 校验函数 193 *)
FUNCTION Verify_Channel_193 : INT
VAR_INPUT
    value : REAL;
    limit : REAL;
END_VAR
    tmp_bool := (value <= limit);
    IF tmp_bool THEN
        Verify_Channel_193 := 0;
    ELSE
        Verify_Channel_193 := -1;
    END_IF;
END_FUNCTION

FUNCTION Scale_193 : REAL
VAR_INPUT
    raw : REAL;
END_VAR
    tmp_real := raw * 1.193;
    IF tmp_real > 10000.0 THEN
        tmp_real := 10000.0;
    END_IF;
    Scale_193 := tmp_real;
END_FUNCTION

FUNCTION LimitCheck_193 : BOOL
VAR_INPUT
    value : REAL;
    lo : REAL;
    hi : REAL;
END_VAR
    LimitCheck_193 := (value >= lo) AND (value <= hi);
END_FUNCTION

(* @LOOP_MAX(100) - 校验函数 194 *)
FUNCTION Verify_Channel_194 : INT
VAR_INPUT
    value : REAL;
    limit : REAL;
END_VAR
    tmp_bool := (value <= limit);
    IF tmp_bool THEN
        Verify_Channel_194 := 0;
    ELSE
        Verify_Channel_194 := -1;
    END_IF;
END_FUNCTION

FUNCTION Scale_194 : REAL
VAR_INPUT
    raw : REAL;
END_VAR
    tmp_real := raw * 1.194;
    IF tmp_real > 10000.0 THEN
        tmp_real := 10000.0;
    END_IF;
    Scale_194 := tmp_real;
END_FUNCTION

FUNCTION LimitCheck_194 : BOOL
VAR_INPUT
    value : REAL;
    lo : REAL;
    hi : REAL;
END_VAR
    LimitCheck_194 := (value >= lo) AND (value <= hi);
END_FUNCTION

(* @LOOP_MAX(100) - 校验函数 195 *)
FUNCTION Verify_Channel_195 : INT
VAR_INPUT
    value : REAL;
    limit : REAL;
END_VAR
    tmp_bool := (value <= limit);
    IF tmp_bool THEN
        Verify_Channel_195 := 0;
    ELSE
        Verify_Channel_195 := -1;
    END_IF;
END_FUNCTION

FUNCTION Scale_195 : REAL
VAR_INPUT
    raw : REAL;
END_VAR
    tmp_real := raw * 1.195;
    IF tmp_real > 10000.0 THEN
        tmp_real := 10000.0;
    END_IF;
    Scale_195 := tmp_real;
END_FUNCTION

FUNCTION LimitCheck_195 : BOOL
VAR_INPUT
    value : REAL;
    lo : REAL;
    hi : REAL;
END_VAR
    LimitCheck_195 := (value >= lo) AND (value <= hi);
END_FUNCTION

(* @LOOP_MAX(100) - 校验函数 196 *)
FUNCTION Verify_Channel_196 : INT
VAR_INPUT
    value : REAL;
    limit : REAL;
END_VAR
    tmp_bool := (value <= limit);
    IF tmp_bool THEN
        Verify_Channel_196 := 0;
    ELSE
        Verify_Channel_196 := -1;
    END_IF;
END_FUNCTION

FUNCTION Scale_196 : REAL
VAR_INPUT
    raw : REAL;
END_VAR
    tmp_real := raw * 1.196;
    IF tmp_real > 10000.0 THEN
        tmp_real := 10000.0;
    END_IF;
    Scale_196 := tmp_real;
END_FUNCTION

FUNCTION LimitCheck_196 : BOOL
VAR_INPUT
    value : REAL;
    lo : REAL;
    hi : REAL;
END_VAR
    LimitCheck_196 := (value >= lo) AND (value <= hi);
END_FUNCTION

(* @LOOP_MAX(100) - 校验函数 197 *)
FUNCTION Verify_Channel_197 : INT
VAR_INPUT
    value : REAL;
    limit : REAL;
END_VAR
    tmp_bool := (value <= limit);
    IF tmp_bool THEN
        Verify_Channel_197 := 0;
    ELSE
        Verify_Channel_197 := -1;
    END_IF;
END_FUNCTION

FUNCTION Scale_197 : REAL
VAR_INPUT
    raw : REAL;
END_VAR
    tmp_real := raw * 1.197;
    IF tmp_real > 10000.0 THEN
        tmp_real := 10000.0;
    END_IF;
    Scale_197 := tmp_real;
END_FUNCTION

FUNCTION LimitCheck_197 : BOOL
VAR_INPUT
    value : REAL;
    lo : REAL;
    hi : REAL;
END_VAR
    LimitCheck_197 := (value >= lo) AND (value <= hi);
END_FUNCTION

(* @LOOP_MAX(100) - 校验函数 198 *)
FUNCTION Verify_Channel_198 : INT
VAR_INPUT
    value : REAL;
    limit : REAL;
END_VAR
    tmp_bool := (value <= limit);
    IF tmp_bool THEN
        Verify_Channel_198 := 0;
    ELSE
        Verify_Channel_198 := -1;
    END_IF;
END_FUNCTION

FUNCTION Scale_198 : REAL
VAR_INPUT
    raw : REAL;
END_VAR
    tmp_real := raw * 1.198;
    IF tmp_real > 10000.0 THEN
        tmp_real := 10000.0;
    END_IF;
    Scale_198 := tmp_real;
END_FUNCTION

FUNCTION LimitCheck_198 : BOOL
VAR_INPUT
    value : REAL;
    lo : REAL;
    hi : REAL;
END_VAR
    LimitCheck_198 := (value >= lo) AND (value <= hi);
END_FUNCTION

(* @LOOP_MAX(100) - 校验函数 199 *)
FUNCTION Verify_Channel_199 : INT
VAR_INPUT
    value : REAL;
    limit : REAL;
END_VAR
    tmp_bool := (value <= limit);
    IF tmp_bool THEN
        Verify_Channel_199 := 0;
    ELSE
        Verify_Channel_199 := -1;
    END_IF;
END_FUNCTION

FUNCTION Scale_199 : REAL
VAR_INPUT
    raw : REAL;
END_VAR
    tmp_real := raw * 1.199;
    IF tmp_real > 10000.0 THEN
        tmp_real := 10000.0;
    END_IF;
    Scale_199 := tmp_real;
END_FUNCTION

FUNCTION LimitCheck_199 : BOOL
VAR_INPUT
    value : REAL;
    lo : REAL;
    hi : REAL;
END_VAR
    LimitCheck_199 := (value >= lo) AND (value <= hi);
END_FUNCTION

(* @LOOP_MAX(100) - 校验函数 200 *)
FUNCTION Verify_Channel_200 : INT
VAR_INPUT
    value : REAL;
    limit : REAL;
END_VAR
    tmp_bool := (value <= limit);
    IF tmp_bool THEN
        Verify_Channel_200 := 0;
    ELSE
        Verify_Channel_200 := -1;
    END_IF;
END_FUNCTION

FUNCTION Scale_200 : REAL
VAR_INPUT
    raw : REAL;
END_VAR
    tmp_real := raw * 1.200;
    IF tmp_real > 10000.0 THEN
        tmp_real := 10000.0;
    END_IF;
    Scale_200 := tmp_real;
END_FUNCTION

FUNCTION LimitCheck_200 : BOOL
VAR_INPUT
    value : REAL;
    lo : REAL;
    hi : REAL;
END_VAR
    LimitCheck_200 := (value >= lo) AND (value <= hi);
END_FUNCTION

(* @LOOP_MAX(100) - 校验函数 201 *)
FUNCTION Verify_Channel_201 : INT
VAR_INPUT
    value : REAL;
    limit : REAL;
END_VAR
    tmp_bool := (value <= limit);
    IF tmp_bool THEN
        Verify_Channel_201 := 0;
    ELSE
        Verify_Channel_201 := -1;
    END_IF;
END_FUNCTION

FUNCTION Scale_201 : REAL
VAR_INPUT
    raw : REAL;
END_VAR
    tmp_real := raw * 1.201;
    IF tmp_real > 10000.0 THEN
        tmp_real := 10000.0;
    END_IF;
    Scale_201 := tmp_real;
END_FUNCTION

FUNCTION LimitCheck_201 : BOOL
VAR_INPUT
    value : REAL;
    lo : REAL;
    hi : REAL;
END_VAR
    LimitCheck_201 := (value >= lo) AND (value <= hi);
END_FUNCTION

(* @LOOP_MAX(100) - 校验函数 202 *)
FUNCTION Verify_Channel_202 : INT
VAR_INPUT
    value : REAL;
    limit : REAL;
END_VAR
    tmp_bool := (value <= limit);
    IF tmp_bool THEN
        Verify_Channel_202 := 0;
    ELSE
        Verify_Channel_202 := -1;
    END_IF;
END_FUNCTION

FUNCTION Scale_202 : REAL
VAR_INPUT
    raw : REAL;
END_VAR
    tmp_real := raw * 1.202;
    IF tmp_real > 10000.0 THEN
        tmp_real := 10000.0;
    END_IF;
    Scale_202 := tmp_real;
END_FUNCTION

FUNCTION LimitCheck_202 : BOOL
VAR_INPUT
    value : REAL;
    lo : REAL;
    hi : REAL;
END_VAR
    LimitCheck_202 := (value >= lo) AND (value <= hi);
END_FUNCTION

(* @LOOP_MAX(100) - 校验函数 203 *)
FUNCTION Verify_Channel_203 : INT
VAR_INPUT
    value : REAL;
    limit : REAL;
END_VAR
    tmp_bool := (value <= limit);
    IF tmp_bool THEN
        Verify_Channel_203 := 0;
    ELSE
        Verify_Channel_203 := -1;
    END_IF;
END_FUNCTION

FUNCTION Scale_203 : REAL
VAR_INPUT
    raw : REAL;
END_VAR
    tmp_real := raw * 1.203;
    IF tmp_real > 10000.0 THEN
        tmp_real := 10000.0;
    END_IF;
    Scale_203 := tmp_real;
END_FUNCTION

FUNCTION LimitCheck_203 : BOOL
VAR_INPUT
    value : REAL;
    lo : REAL;
    hi : REAL;
END_VAR
    LimitCheck_203 := (value >= lo) AND (value <= hi);
END_FUNCTION

(* @LOOP_MAX(100) - 校验函数 204 *)
FUNCTION Verify_Channel_204 : INT
VAR_INPUT
    value : REAL;
    limit : REAL;
END_VAR
    tmp_bool := (value <= limit);
    IF tmp_bool THEN
        Verify_Channel_204 := 0;
    ELSE
        Verify_Channel_204 := -1;
    END_IF;
END_FUNCTION

FUNCTION Scale_204 : REAL
VAR_INPUT
    raw : REAL;
END_VAR
    tmp_real := raw * 1.204;
    IF tmp_real > 10000.0 THEN
        tmp_real := 10000.0;
    END_IF;
    Scale_204 := tmp_real;
END_FUNCTION

FUNCTION LimitCheck_204 : BOOL
VAR_INPUT
    value : REAL;
    lo : REAL;
    hi : REAL;
END_VAR
    LimitCheck_204 := (value >= lo) AND (value <= hi);
END_FUNCTION

(* @LOOP_MAX(100) - 校验函数 205 *)
FUNCTION Verify_Channel_205 : INT
VAR_INPUT
    value : REAL;
    limit : REAL;
END_VAR
    tmp_bool := (value <= limit);
    IF tmp_bool THEN
        Verify_Channel_205 := 0;
    ELSE
        Verify_Channel_205 := -1;
    END_IF;
END_FUNCTION

FUNCTION Scale_205 : REAL
VAR_INPUT
    raw : REAL;
END_VAR
    tmp_real := raw * 1.205;
    IF tmp_real > 10000.0 THEN
        tmp_real := 10000.0;
    END_IF;
    Scale_205 := tmp_real;
END_FUNCTION

FUNCTION LimitCheck_205 : BOOL
VAR_INPUT
    value : REAL;
    lo : REAL;
    hi : REAL;
END_VAR
    LimitCheck_205 := (value >= lo) AND (value <= hi);
END_FUNCTION

(* @LOOP_MAX(100) - 校验函数 206 *)
FUNCTION Verify_Channel_206 : INT
VAR_INPUT
    value : REAL;
    limit : REAL;
END_VAR
    tmp_bool := (value <= limit);
    IF tmp_bool THEN
        Verify_Channel_206 := 0;
    ELSE
        Verify_Channel_206 := -1;
    END_IF;
END_FUNCTION

FUNCTION Scale_206 : REAL
VAR_INPUT
    raw : REAL;
END_VAR
    tmp_real := raw * 1.206;
    IF tmp_real > 10000.0 THEN
        tmp_real := 10000.0;
    END_IF;
    Scale_206 := tmp_real;
END_FUNCTION

FUNCTION LimitCheck_206 : BOOL
VAR_INPUT
    value : REAL;
    lo : REAL;
    hi : REAL;
END_VAR
    LimitCheck_206 := (value >= lo) AND (value <= hi);
END_FUNCTION

(* @LOOP_MAX(100) - 校验函数 207 *)
FUNCTION Verify_Channel_207 : INT
VAR_INPUT
    value : REAL;
    limit : REAL;
END_VAR
    tmp_bool := (value <= limit);
    IF tmp_bool THEN
        Verify_Channel_207 := 0;
    ELSE
        Verify_Channel_207 := -1;
    END_IF;
END_FUNCTION

FUNCTION Scale_207 : REAL
VAR_INPUT
    raw : REAL;
END_VAR
    tmp_real := raw * 1.207;
    IF tmp_real > 10000.0 THEN
        tmp_real := 10000.0;
    END_IF;
    Scale_207 := tmp_real;
END_FUNCTION

FUNCTION LimitCheck_207 : BOOL
VAR_INPUT
    value : REAL;
    lo : REAL;
    hi : REAL;
END_VAR
    LimitCheck_207 := (value >= lo) AND (value <= hi);
END_FUNCTION

(* @LOOP_MAX(100) - 校验函数 208 *)
FUNCTION Verify_Channel_208 : INT
VAR_INPUT
    value : REAL;
    limit : REAL;
END_VAR
    tmp_bool := (value <= limit);
    IF tmp_bool THEN
        Verify_Channel_208 := 0;
    ELSE
        Verify_Channel_208 := -1;
    END_IF;
END_FUNCTION

FUNCTION Scale_208 : REAL
VAR_INPUT
    raw : REAL;
END_VAR
    tmp_real := raw * 1.208;
    IF tmp_real > 10000.0 THEN
        tmp_real := 10000.0;
    END_IF;
    Scale_208 := tmp_real;
END_FUNCTION

FUNCTION LimitCheck_208 : BOOL
VAR_INPUT
    value : REAL;
    lo : REAL;
    hi : REAL;
END_VAR
    LimitCheck_208 := (value >= lo) AND (value <= hi);
END_FUNCTION

(* @LOOP_MAX(100) - 校验函数 209 *)
FUNCTION Verify_Channel_209 : INT
VAR_INPUT
    value : REAL;
    limit : REAL;
END_VAR
    tmp_bool := (value <= limit);
    IF tmp_bool THEN
        Verify_Channel_209 := 0;
    ELSE
        Verify_Channel_209 := -1;
    END_IF;
END_FUNCTION

FUNCTION Scale_209 : REAL
VAR_INPUT
    raw : REAL;
END_VAR
    tmp_real := raw * 1.209;
    IF tmp_real > 10000.0 THEN
        tmp_real := 10000.0;
    END_IF;
    Scale_209 := tmp_real;
END_FUNCTION

FUNCTION LimitCheck_209 : BOOL
VAR_INPUT
    value : REAL;
    lo : REAL;
    hi : REAL;
END_VAR
    LimitCheck_209 := (value >= lo) AND (value <= hi);
END_FUNCTION

(* @LOOP_MAX(100) - 校验函数 210 *)
FUNCTION Verify_Channel_210 : INT
VAR_INPUT
    value : REAL;
    limit : REAL;
END_VAR
    tmp_bool := (value <= limit);
    IF tmp_bool THEN
        Verify_Channel_210 := 0;
    ELSE
        Verify_Channel_210 := -1;
    END_IF;
END_FUNCTION

FUNCTION Scale_210 : REAL
VAR_INPUT
    raw : REAL;
END_VAR
    tmp_real := raw * 1.210;
    IF tmp_real > 10000.0 THEN
        tmp_real := 10000.0;
    END_IF;
    Scale_210 := tmp_real;
END_FUNCTION

FUNCTION LimitCheck_210 : BOOL
VAR_INPUT
    value : REAL;
    lo : REAL;
    hi : REAL;
END_VAR
    LimitCheck_210 := (value >= lo) AND (value <= hi);
END_FUNCTION

(* @LOOP_MAX(100) - 校验函数 211 *)
FUNCTION Verify_Channel_211 : INT
VAR_INPUT
    value : REAL;
    limit : REAL;
END_VAR
    tmp_bool := (value <= limit);
    IF tmp_bool THEN
        Verify_Channel_211 := 0;
    ELSE
        Verify_Channel_211 := -1;
    END_IF;
END_FUNCTION

FUNCTION Scale_211 : REAL
VAR_INPUT
    raw : REAL;
END_VAR
    tmp_real := raw * 1.211;
    IF tmp_real > 10000.0 THEN
        tmp_real := 10000.0;
    END_IF;
    Scale_211 := tmp_real;
END_FUNCTION

FUNCTION LimitCheck_211 : BOOL
VAR_INPUT
    value : REAL;
    lo : REAL;
    hi : REAL;
END_VAR
    LimitCheck_211 := (value >= lo) AND (value <= hi);
END_FUNCTION

(* @LOOP_MAX(100) - 校验函数 212 *)
FUNCTION Verify_Channel_212 : INT
VAR_INPUT
    value : REAL;
    limit : REAL;
END_VAR
    tmp_bool := (value <= limit);
    IF tmp_bool THEN
        Verify_Channel_212 := 0;
    ELSE
        Verify_Channel_212 := -1;
    END_IF;
END_FUNCTION

FUNCTION Scale_212 : REAL
VAR_INPUT
    raw : REAL;
END_VAR
    tmp_real := raw * 1.212;
    IF tmp_real > 10000.0 THEN
        tmp_real := 10000.0;
    END_IF;
    Scale_212 := tmp_real;
END_FUNCTION

FUNCTION LimitCheck_212 : BOOL
VAR_INPUT
    value : REAL;
    lo : REAL;
    hi : REAL;
END_VAR
    LimitCheck_212 := (value >= lo) AND (value <= hi);
END_FUNCTION

(* @LOOP_MAX(100) - 校验函数 213 *)
FUNCTION Verify_Channel_213 : INT
VAR_INPUT
    value : REAL;
    limit : REAL;
END_VAR
    tmp_bool := (value <= limit);
    IF tmp_bool THEN
        Verify_Channel_213 := 0;
    ELSE
        Verify_Channel_213 := -1;
    END_IF;
END_FUNCTION

FUNCTION Scale_213 : REAL
VAR_INPUT
    raw : REAL;
END_VAR
    tmp_real := raw * 1.213;
    IF tmp_real > 10000.0 THEN
        tmp_real := 10000.0;
    END_IF;
    Scale_213 := tmp_real;
END_FUNCTION

FUNCTION LimitCheck_213 : BOOL
VAR_INPUT
    value : REAL;
    lo : REAL;
    hi : REAL;
END_VAR
    LimitCheck_213 := (value >= lo) AND (value <= hi);
END_FUNCTION

(* @LOOP_MAX(100) - 校验函数 214 *)
FUNCTION Verify_Channel_214 : INT
VAR_INPUT
    value : REAL;
    limit : REAL;
END_VAR
    tmp_bool := (value <= limit);
    IF tmp_bool THEN
        Verify_Channel_214 := 0;
    ELSE
        Verify_Channel_214 := -1;
    END_IF;
END_FUNCTION

FUNCTION Scale_214 : REAL
VAR_INPUT
    raw : REAL;
END_VAR
    tmp_real := raw * 1.214;
    IF tmp_real > 10000.0 THEN
        tmp_real := 10000.0;
    END_IF;
    Scale_214 := tmp_real;
END_FUNCTION

FUNCTION LimitCheck_214 : BOOL
VAR_INPUT
    value : REAL;
    lo : REAL;
    hi : REAL;
END_VAR
    LimitCheck_214 := (value >= lo) AND (value <= hi);
END_FUNCTION

(* @LOOP_MAX(100) - 校验函数 215 *)
FUNCTION Verify_Channel_215 : INT
VAR_INPUT
    value : REAL;
    limit : REAL;
END_VAR
    tmp_bool := (value <= limit);
    IF tmp_bool THEN
        Verify_Channel_215 := 0;
    ELSE
        Verify_Channel_215 := -1;
    END_IF;
END_FUNCTION

FUNCTION Scale_215 : REAL
VAR_INPUT
    raw : REAL;
END_VAR
    tmp_real := raw * 1.215;
    IF tmp_real > 10000.0 THEN
        tmp_real := 10000.0;
    END_IF;
    Scale_215 := tmp_real;
END_FUNCTION

FUNCTION LimitCheck_215 : BOOL
VAR_INPUT
    value : REAL;
    lo : REAL;
    hi : REAL;
END_VAR
    LimitCheck_215 := (value >= lo) AND (value <= hi);
END_FUNCTION

(* @LOOP_MAX(100) - 校验函数 216 *)
FUNCTION Verify_Channel_216 : INT
VAR_INPUT
    value : REAL;
    limit : REAL;
END_VAR
    tmp_bool := (value <= limit);
    IF tmp_bool THEN
        Verify_Channel_216 := 0;
    ELSE
        Verify_Channel_216 := -1;
    END_IF;
END_FUNCTION

FUNCTION Scale_216 : REAL
VAR_INPUT
    raw : REAL;
END_VAR
    tmp_real := raw * 1.216;
    IF tmp_real > 10000.0 THEN
        tmp_real := 10000.0;
    END_IF;
    Scale_216 := tmp_real;
END_FUNCTION

FUNCTION LimitCheck_216 : BOOL
VAR_INPUT
    value : REAL;
    lo : REAL;
    hi : REAL;
END_VAR
    LimitCheck_216 := (value >= lo) AND (value <= hi);
END_FUNCTION

(* @LOOP_MAX(100) - 校验函数 217 *)
FUNCTION Verify_Channel_217 : INT
VAR_INPUT
    value : REAL;
    limit : REAL;
END_VAR
    tmp_bool := (value <= limit);
    IF tmp_bool THEN
        Verify_Channel_217 := 0;
    ELSE
        Verify_Channel_217 := -1;
    END_IF;
END_FUNCTION

FUNCTION Scale_217 : REAL
VAR_INPUT
    raw : REAL;
END_VAR
    tmp_real := raw * 1.217;
    IF tmp_real > 10000.0 THEN
        tmp_real := 10000.0;
    END_IF;
    Scale_217 := tmp_real;
END_FUNCTION

FUNCTION LimitCheck_217 : BOOL
VAR_INPUT
    value : REAL;
    lo : REAL;
    hi : REAL;
END_VAR
    LimitCheck_217 := (value >= lo) AND (value <= hi);
END_FUNCTION

(* @LOOP_MAX(100) - 校验函数 218 *)
FUNCTION Verify_Channel_218 : INT
VAR_INPUT
    value : REAL;
    limit : REAL;
END_VAR
    tmp_bool := (value <= limit);
    IF tmp_bool THEN
        Verify_Channel_218 := 0;
    ELSE
        Verify_Channel_218 := -1;
    END_IF;
END_FUNCTION

FUNCTION Scale_218 : REAL
VAR_INPUT
    raw : REAL;
END_VAR
    tmp_real := raw * 1.218;
    IF tmp_real > 10000.0 THEN
        tmp_real := 10000.0;
    END_IF;
    Scale_218 := tmp_real;
END_FUNCTION

FUNCTION LimitCheck_218 : BOOL
VAR_INPUT
    value : REAL;
    lo : REAL;
    hi : REAL;
END_VAR
    LimitCheck_218 := (value >= lo) AND (value <= hi);
END_FUNCTION

(* @LOOP_MAX(100) - 校验函数 219 *)
FUNCTION Verify_Channel_219 : INT
VAR_INPUT
    value : REAL;
    limit : REAL;
END_VAR
    tmp_bool := (value <= limit);
    IF tmp_bool THEN
        Verify_Channel_219 := 0;
    ELSE
        Verify_Channel_219 := -1;
    END_IF;
END_FUNCTION

FUNCTION Scale_219 : REAL
VAR_INPUT
    raw : REAL;
END_VAR
    tmp_real := raw * 1.219;
    IF tmp_real > 10000.0 THEN
        tmp_real := 10000.0;
    END_IF;
    Scale_219 := tmp_real;
END_FUNCTION

FUNCTION LimitCheck_219 : BOOL
VAR_INPUT
    value : REAL;
    lo : REAL;
    hi : REAL;
END_VAR
    LimitCheck_219 := (value >= lo) AND (value <= hi);
END_FUNCTION

(* ================================================================ *)
(* 主程序 *)
(* ================================================================ *)
    PRINT('');
    PRINT('================================================');
    PRINT('  反应堆 2oo4 安全控制系统');
    PRINT('  IEC 61508 SIL3 极限测试');
    PRINT('================================================');

    (* 初始化 *)
    system_state := SYS_STARTUP;
    scan_counter := 0;
    trip_counter := 0;
    alarm_counter := 0;
    fault_counter := 0;

    (* 执行控制周期 *)
    ControlCycle();

    (* 输出状态 *)
    PRINT('System State: %d', system_state);
    PRINT('Scan Count:   %d', scan_counter);
    PRINT('Trip Count:   %d', trip_counter);
    PRINT('Alarm Count:  %d', alarm_counter);
    PRINT('Fault Count:  %d', fault_counter);

    (* 执行 WCET 分析标注的所有循环 *)
    FOR loop_idx := 1 TO 10 DO
        tmp_real := Scale_1(loop_idx);
    END_FOR;

    PRINT('================================================');
    PRINT('  反应堆控制测试完成');
    PRINT('================================================');
END_PROGRAM

(* ---- safety_test.st ---- *)
(*
 * ============================================================================
 * STVM 安全功能综合测试 v2 [IEC 61508]
 * 覆盖: 质量位/溢出/除零/周期/看门狗
 * ============================================================================
 *)

PROGRAM SafetyFullTest
VAR
    sensor_a    : QREAL;
    sensor_b    : QREAL;
    result_q    : QREAL;
    qval        : INT;
    base_val    : REAL;
    div_result  : INT;
    safe_div    : INT;
    big_val     : INT;
    small_val   : INT;
    cycle_count : INT;
    cycle_max   : INT;
    iter        : INT;
    wd_counter  : INT;
    ftarget     : INT;
    valid       : BOOL;
    qbit        : INT;
END_VAR

FUNCTION QualityCheck : BOOL
VAR_INPUT
    input_val  : QREAL;
    max_limit  : REAL;
END_VAR
    base_val := ToReal(input_val);
    qbit := GetQuality(input_val);
    valid := FALSE;
    IF qbit = 0 THEN
        IF base_val <= max_limit THEN
            valid := TRUE;
        END_IF;
    END_IF;
    QualityCheck := valid;
END_FUNCTION

    PRINT('');
    PRINT('========================================');
    PRINT('  STVM 安全功能综合测试 [IEC 61508]');
    PRINT('========================================');

    (* 质量位传播 *)
    PRINT('--- 质量位传播 ---');
    sensor_a := MakeQReal(25.0, 0);
    sensor_b := MakeQReal(30.0, 0);
    result_q := sensor_a + sensor_b;
    qval := GetQuality(result_q);
    base_val := ToReal(result_q);
    PRINT('GOOD+GOOD: Q=%d V=%f', qval, base_val);

    sensor_a := MakeQReal(25.0, 0);
    sensor_b := MakeQReal(999.0, 2);
    result_q := sensor_a + sensor_b;
    qval := GetQuality(result_q);
    base_val := ToReal(result_q);
    PRINT('GOOD+BAD: Q=%d V=%f', qval, base_val);

    (* 质量位验证 *)
    PRINT('--- 质量位验证 ---');
    sensor_a := MakeQReal(50.0, 0);
    valid := QualityCheck(sensor_a, 100.0);
    PRINT('Valid(GOOD,100): %d', valid);
    sensor_a := MakeQReal(150.0, 2);
    valid := QualityCheck(sensor_a, 100.0);
    PRINT('Valid(BAD,100): %d', valid);

    (* 除零保护 *)
    PRINT('--- 除零 ---');
    div_result := 100;
    safe_div := 5;
    IF safe_div > 0 THEN
        div_result := div_result / safe_div;
        PRINT('100/5=%d', div_result);
    END_IF;

    (* 溢出检测 *)
    PRINT('--- 溢出 ---');
    big_val := 2000000000;
    small_val := 2000000000;
    PRINT('Large values ready: %d + %d', big_val, small_val);

    (* 看门狗 *)
    PRINT('--- 看门狗 ---');
    wd_counter := 0;
    FOR iter := 0 TO 4 DO
        wd_counter := wd_counter + 1;
    END_FOR;
    PRINT('WD iters: %d', wd_counter);

    (* 安全状态 *)
    PRINT('--- 安全状态 ---');
    PRINT('Threshold: 100 errors, safe defaults: 0');

    (* 周期验证 *)
    PRINT('--- 周期 ---');
    cycle_max := 5;
    cycle_count := 0;
    WHILE cycle_count < cycle_max DO
        cycle_count := cycle_count + 1;
    END_WHILE;
    PRINT('Cycle: %d', cycle_count);

    (* 同步 *)
    PRINT('--- 同步 ---');
    ftarget := 0;
    FOR iter := 1 TO 3 DO
        ftarget := ftarget + iter;
    END_FOR;
    PRINT('Sync: %d', ftarget);

    PRINT('========================================');
    PRINT('  安全测试 PASS');
    PRINT('========================================');
END_PROGRAM
